gfCNCPoint4[26389] = {X -0.0949, Y 100.0187, Z -6.3333, A 0.000, B 0.000, C 0.000 }
gfCNCPoint4[26390] = {X -0.0672, Y 100.0699, Z -6.3333, A 0.000, B 0.000, C 0.000 }
gfCNCPoint4[26391] = {X -0.0148, Y 100.0951, Z -6.3333, A 0.000, B 0.000, C 0.000 }
gfCNCPoint4[26392] = {X 120.5926, Y 100.0951, Z -6.3333, A 0.000, B 0.000, C 0.000 }
gfCNCPoint4[26393] = {X 121.0614, Y 100.8813, Z -6.3333, A 0.000, B 0.000, C 0.000 }
gfCNCPoint4[26394] = {X 121.6687, Y 101.5661, Z -6.3333, A 0.000, B 0.000, C 0.000 }
gfCNCPoint4[26395] = {X 122.3932, Y 102.1254, Z -6.3333, A 0.000, B 0.000, C 0.000 }
gfCNCPoint4[26396] = {X 123.2095, Y 102.5397, Z -6.3333, A 0.000, B 0.000, C 0.000 }
gfCNCPoint4[26397] = {X 124.0887, Y 102.7942, Z -6.3333, A 0.000, B 0.000, C 0.000 }
gfCNCPoint4[26398] = {X 125.0000, Y 102.8800, Z -6.3333, A 0.000, B 0.000, C 0.000 }
gfCNCPoint4[26399] = {X 143.7791, Y 102.8800, Z -6.3333, A 0.000, B 0.000, C 0.000 }
gfCNCPoint4[26400] = {X 144.6904, Y 102.7942, Z -6.3333, A 0.000, B 0.000, C 0.000 }
gfCNCPoint4[26401] = {X 145.5696, Y 102.5397, Z -6.3333, A 0.000, B 0.000, C 0.000 }
gfCNCPoint4[26402] = {X 146.3859, Y 102.1254, Z -6.3333, A 0.000, B 0.000, C 0.000 }
gfCNCPoint4[26403] = {X 147.1104, Y 101.5661, Z -6.3333, A 0.000, B 0.000, C 0.000 }
gfCNCPoint4[26404] = {X 147.7177, Y 100.8813, Z -6.3333, A 0.000, B 0.000, C 0.000 }
gfCNCPoint4[26405] = {X 148.1865, Y 100.0951, Z -6.3333, A 0.000, B 0.000, C 0.000 }
gfCNCPoint4[26406] = {X 150.8385, Y 100.0951, Z -6.3333, A 0.000, B 0.000, C 0.000 }
gfCNCPoint4[26407] = {X 150.8385, Y 95.2951, Z -6.3333, A 0.000, B 0.000, C 0.000 }
gfCNCPoint4[26408] = {X 187.9256, Y 95.2951, Z -6.3333, A 0.000, B 0.000, C 0.000 }
gfCNCPoint4[26409] = {X 187.9777, Y 95.0990, Z -6.3333, A 0.000, B 0.000, C 0.000 }
gfCNCPoint4[26410] = {X 188.0352, Y 94.9045, Z -6.3333, A 0.000, B 0.000, C 0.000 }
gfCNCPoint4[26411] = {X 187.2619, Y 94.0602, Z -6.3333, A 0.000, B 0.000, C 0.000 }
gfCNCPoint4[26412] = {X 151.4055, Y 94.0602, Z -6.3333, A 0.000, B 0.000, C 0.000 }
gfCNCPoint4[26413] = {X 150.7064, Y 94.8347, Z -6.3333, A 0.000, B 0.000, C 0.000 }
gfCNCPoint4[26414] = {X 150.7762, Y 95.0638, Z -6.3333, A 0.000, B 0.000, C 0.000 }
gfCNCPoint4[26415] = {X 150.8385, Y 95.2951, Z -6.3333, A 0.000, B 0.000, C 0.000 }
gfCNCPoint4[26416] = {X 150.8385, Y 97.6951, Z -6.3333, A 0.000, B 0.000, C 0.000 }
gfCNCPoint4[26417] = {X 190.1070, Y 97.6951, Z -6.3333, A 0.000, B 0.000, C 0.000 }
gfCNCPoint4[26418] = {X 190.1070, Y 97.0659, Z -6.3333, A 0.000, B 0.000, C 0.000 }
gfCNCPoint4[26419] = {X 190.1938, Y 96.1495, Z -6.3333, A 0.000, B 0.000, C 0.000 }
gfCNCPoint4[26420] = {X 190.4511, Y 95.2657, Z -6.3333, A 0.000, B 0.000, C 0.000 }
gfCNCPoint4[26421] = {X 190.8699, Y 94.4460, Z -6.3333, A 0.000, B 0.000, C 0.000 }
gfCNCPoint4[26422] = {X 188.3182, Y 91.6602, Z -6.3333, A 0.000, B 0.000, C 0.000 }
gfCNCPoint4[26423] = {X 150.3387, Y 91.6602, Z -6.3333, A 0.000, B 0.000, C 0.000 }
gfCNCPoint4[26424] = {X 147.8644, Y 94.4015, Z -6.3333, A 0.000, B 0.000, C 0.000 }
gfCNCPoint4[26425] = {X 148.2989, Y 95.2324, Z -6.3333, A 0.000, B 0.000, C 0.000 }
gfCNCPoint4[26426] = {X 148.5670, Y 96.1308, Z -6.3333, A 0.000, B 0.000, C 0.000 }
gfCNCPoint4[26427] = {X 148.6591, Y 97.0639, Z -6.3333, A 0.000, B 0.000, C 0.000 }
gfCNCPoint4[26428] = {X 148.6591, Y 97.6951, Z -6.3333, A 0.000, B 0.000, C 0.000 }
gfCNCPoint4[26429] = {X 150.8385, Y 97.6951, Z -6.3333, A 0.000, B 0.000, C 0.000 }
gfCNCPoint4[26430] = {X 150.8385, Y 100.0951, Z -6.3333, A 0.000, B 0.000, C 0.000 }
gfCNCPoint4[26431] = {X 190.5796, Y 100.0951, Z -6.3333, A 0.000, B 0.000, C 0.000 }
gfCNCPoint4[26432] = {X 191.0483, Y 100.8813, Z -6.3333, A 0.000, B 0.000, C 0.000 }
gfCNCPoint4[26433] = {X 191.6557, Y 101.5661, Z -6.3333, A 0.000, B 0.000, C 0.000 }
gfCNCPoint4[26434] = {X 192.3802, Y 102.1254, Z -6.3333, A 0.000, B 0.000, C 0.000 }
gfCNCPoint4[26435] = {X 193.1964, Y 102.5397, Z -6.3333, A 0.000, B 0.000, C 0.000 }
gfCNCPoint4[26436] = {X 194.0757, Y 102.7942, Z -6.3333, A 0.000, B 0.000, C 0.000 }
gfCNCPoint4[26437] = {X 194.9870, Y 102.8800, Z -6.3333, A 0.000, B 0.000, C 0.000 }
gfCNCPoint4[26438] = {X 212.6141, Y 102.8800, Z -6.3333, A 0.000, B 0.000, C 0.000 }
gfCNCPoint4[26439] = {X 213.0066, Y 102.8642, Z -6.3333, A 0.000, B 0.000, C 0.000 }
gfCNCPoint4[26440] = {X 213.3966, Y 102.8169, Z -6.3333, A 0.000, B 0.000, C 0.000 }
gfCNCPoint4[26441] = {X 213.7865, Y 102.8642, Z -6.3333, A 0.000, B 0.000, C 0.000 }
gfCNCPoint4[26442] = {X 214.1790, Y 102.8800, Z -6.3333, A 0.000, B 0.000, C 0.000 }
gfCNCPoint4[26443] = {X 233.4798, Y 102.8800, Z -6.3333, A 0.000, B 0.000, C 0.000 }
gfCNCPoint4[26444] = {X 234.3911, Y 102.7942, Z -6.3333, A 0.000, B 0.000, C 0.000 }
gfCNCPoint4[26445] = {X 235.2703, Y 102.5397, Z -6.3333, A 0.000, B 0.000, C 0.000 }
gfCNCPoint4[26446] = {X 236.0865, Y 102.1254, Z -6.3333, A 0.000, B 0.000, C 0.000 }
gfCNCPoint4[26447] = {X 236.8111, Y 101.5661, Z -6.3333, A 0.000, B 0.000, C 0.000 }
gfCNCPoint4[26448] = {X 237.4184, Y 100.8813, Z -6.3333, A 0.000, B 0.000, C 0.000 }
gfCNCPoint4[26449] = {X 237.8872, Y 100.0951, Z -6.3333, A 0.000, B 0.000, C 0.000 }
gfCNCPoint4[26450] = {X 261.4782, Y 100.0951, Z -6.3333, A 0.000, B 0.000, C 0.000 }
gfCNCPoint4[26451] = {X 261.4782, Y 90.4951, Z -6.3333, A 0.000, B 0.000, C 0.000 }
gfCNCPoint4[26452] = {X 266.0961, Y 90.4951, Z -6.3333, A 0.000, B 0.000, C 0.000 }
gfCNCPoint4[26453] = {X 266.1751, Y 90.3748, Z -6.3333, A 0.000, B 0.000, C 0.000 }
gfCNCPoint4[26454] = {X 266.2556, Y 90.2554, Z -6.3333, A 0.000, B 0.000, C 0.000 }
gfCNCPoint4[26455] = {X 263.5100, Y 89.1791, Z -6.3333, A 0.000, B 0.000, C 0.000 }
gfCNCPoint4[26456] = {X 261.4782, Y 90.4951, Z -6.3333, A 0.000, B 0.000, C 0.000 }
gfCNCPoint4[26457] = {X 261.4782, Y 92.8951, Z -6.3333, A 0.000, B 0.000, C 0.000 }
gfCNCPoint4[26458] = {X 267.4973, Y 92.8951, Z -6.3333, A 0.000, B 0.000, C 0.000 }
gfCNCPoint4[26459] = {X 267.8429, Y 92.2376, Z -6.3333, A 0.000, B 0.000, C 0.000 }
gfCNCPoint4[26460] = {X 268.2378, Y 91.6085, Z -6.3333, A 0.000, B 0.000, C 0.000 }
gfCNCPoint4[26461] = {X 269.1700, Y 90.4463, Z -6.3333, A 0.000, B 0.000, C 0.000 }
gfCNCPoint4[26462] = {X 270.2694, Y 89.4409, Z -6.3333, A 0.000, B 0.000, C 0.000 }
gfCNCPoint4[26463] = {X 270.2694, Y 89.2510, Z -6.3333, A 0.000, B 0.000, C 0.000 }
gfCNCPoint4[26464] = {X 263.2391, Y 86.4951, Z -6.3333, A 0.000, B 0.000, C 0.000 }
gfCNCPoint4[26465] = {X 253.3583, Y 92.8951, Z -6.3333, A 0.000, B 0.000, C 0.000 }
gfCNCPoint4[26466] = {X 261.4782, Y 92.8951, Z -6.3333, A 0.000, B 0.000, C 0.000 }
gfCNCPoint4[26467] = {X 261.4782, Y 95.2951, Z -6.3333, A 0.000, B 0.000, C 0.000 }
gfCNCPoint4[26468] = {X 269.1714, Y 95.2951, Z -6.3333, A 0.000, B 0.000, C 0.000 }
gfCNCPoint4[26469] = {X 269.5515, Y 94.1745, Z -6.3333, A 0.000, B 0.000, C 0.000 }
gfCNCPoint4[26470] = {X 270.1082, Y 93.1303, Z -6.3333, A 0.000, B 0.000, C 0.000 }
gfCNCPoint4[26471] = {X 270.8267, Y 92.1901, Z -6.3333, A 0.000, B 0.000, C 0.000 }
gfCNCPoint4[26472] = {X 271.6880, Y 91.3787, Z -6.3333, A 0.000, B 0.000, C 0.000 }
gfCNCPoint4[26473] = {X 272.6694, Y 90.7176, Z -6.3333, A 0.000, B 0.000, C 0.000 }
gfCNCPoint4[26474] = {X 272.6694, Y 87.6139, Z -6.3333, A 0.000, B 0.000, C 0.000 }
gfCNCPoint4[26475] = {X 262.9682, Y 83.8111, Z -6.3333, A 0.000, B 0.000, C 0.000 }
gfCNCPoint4[26476] = {X 245.2384, Y 95.2951, Z -6.3333, A 0.000, B 0.000, C 0.000 }
gfCNCPoint4[26477] = {X 261.4782, Y 95.2951, Z -6.3333, A 0.000, B 0.000, C 0.000 }
gfCNCPoint4[26478] = {X 261.4782, Y 97.6951, Z -6.3333, A 0.000, B 0.000, C 0.000 }
gfCNCPoint4[26479] = {X 271.3527, Y 97.6951, Z -6.3333, A 0.000, B 0.000, C 0.000 }
gfCNCPoint4[26480] = {X 271.3529, Y 97.0186, Z -6.3333, A 0.000, B 0.000, C 0.000 }
gfCNCPoint4[26481] = {X 271.4810, Y 95.9545, Z -6.3333, A 0.000, B 0.000, C 0.000 }
gfCNCPoint4[26482] = {X 271.8382, Y 94.9440, Z -6.3333, A 0.000, B 0.000, C 0.000 }
gfCNCPoint4[26483] = {X 272.4073, Y 94.0359, Z -6.3333, A 0.000, B 0.000, C 0.000 }
gfCNCPoint4[26484] = {X 273.1610, Y 93.2739, Z -6.3333, A 0.000, B 0.000, C 0.000 }
gfCNCPoint4[26485] = {X 274.0629, Y 92.6949, Z -6.3333, A 0.000, B 0.000, C 0.000 }
gfCNCPoint4[26486] = {X 275.0694, Y 92.3266, Z -6.3333, A 0.000, B 0.000, C 0.000 }
gfCNCPoint4[26487] = {X 275.0694, Y 85.9769, Z -6.3333, A 0.000, B 0.000, C 0.000 }
gfCNCPoint4[26488] = {X 262.6992, Y 81.1278, Z -6.3333, A 0.000, B 0.000, C 0.000 }
gfCNCPoint4[26489] = {X 262.5795, Y 81.2034, Z -6.3333, A 0.000, B 0.000, C 0.000 }
gfCNCPoint4[26490] = {X 238.3588, Y 96.8917, Z -6.3333, A 0.000, B 0.000, C 0.000 }
gfCNCPoint4[26491] = {X 238.3598, Y 97.0659, Z -6.3333, A 0.000, B 0.000, C 0.000 }
gfCNCPoint4[26492] = {X 238.3598, Y 97.6951, Z -6.3333, A 0.000, B 0.000, C 0.000 }
gfCNCPoint4[26493] = {X 261.4782, Y 97.6951, Z -6.3333, A 0.000, B 0.000, C 0.000 }
gfCNCPoint4[26494] = {X 261.4782, Y 100.0951, Z -6.3333, A 0.000, B 0.000, C 0.000 }
gfCNCPoint4[26495] = {X 271.8253, Y 100.0951, Z -6.3333, A 0.000, B 0.000, C 0.000 }
gfCNCPoint4[26496] = {X 272.2941, Y 100.8813, Z -6.3333, A 0.000, B 0.000, C 0.000 }
gfCNCPoint4[26497] = {X 272.9014, Y 101.5661, Z -6.3333, A 0.000, B 0.000, C 0.000 }
gfCNCPoint4[26498] = {X 273.6259, Y 102.1254, Z -6.3333, A 0.000, B 0.000, C 0.000 }
gfCNCPoint4[26499] = {X 274.4422, Y 102.5397, Z -6.3333, A 0.000, B 0.000, C 0.000 }
gfCNCPoint4[26500] = {X 275.3214, Y 102.7942, Z -6.3333, A 0.000, B 0.000, C 0.000 }
gfCNCPoint4[26501] = {X 276.2327, Y 102.8800, Z -6.3333, A 0.000, B 0.000, C 0.000 }
gfCNCPoint4[26502] = {X 292.7731, Y 102.8800, Z -6.3333, A 0.000, B 0.000, C 0.000 }
gfCNCPoint4[26503] = {X 293.6844, Y 102.7942, Z -6.3333, A 0.000, B 0.000, C 0.000 }
gfCNCPoint4[26504] = {X 294.5636, Y 102.5397, Z -6.3333, A 0.000, B 0.000, C 0.000 }
gfCNCPoint4[26505] = {X 295.3798, Y 102.1254, Z -6.3333, A 0.000, B 0.000, C 0.000 }
gfCNCPoint4[26506] = {X 296.1044, Y 101.5661, Z -6.3333, A 0.000, B 0.000, C 0.000 }
gfCNCPoint4[26507] = {X 296.7117, Y 100.8813, Z -6.3333, A 0.000, B 0.000, C 0.000 }
gfCNCPoint4[26508] = {X 297.1805, Y 100.0951, Z -6.3333, A 0.000, B 0.000, C 0.000 }
gfCNCPoint4[26509] = {X 319.1325, Y 100.0951, Z -6.3333, A 0.000, B 0.000, C 0.000 }
gfCNCPoint4[26510] = {X 321.4361, Y 100.8683, Z -6.3333, A 0.000, B 0.000, C 0.000 }
gfCNCPoint4[26511] = {X 323.7823, Y 101.5005, Z -6.3333, A 0.000, B 0.000, C 0.000 }
gfCNCPoint4[26512] = {X 326.1626, Y 101.9893, Z -6.3333, A 0.000, B 0.000, C 0.000 }
gfCNCPoint4[26513] = {X 330.1025, Y 102.5988, Z -6.3333, A 0.000, B 0.000, C 0.000 }
gfCNCPoint4[26514] = {X 334.0644, Y 103.0432, Z -6.3333, A 0.000, B 0.000, C 0.000 }
gfCNCPoint4[26515] = {X 338.0414, Y 103.3217, Z -6.3333, A 0.000, B 0.000, C 0.000 }
gfCNCPoint4[26516] = {X 343.7798, Y 103.5423, Z -6.3333, A 0.000, B 0.000, C 0.000 }
gfCNCPoint4[26517] = {X 349.5223, Y 103.5874, Z -6.3333, A 0.000, B 0.000, C 0.000 }
gfCNCPoint4[26518] = {X 355.2635, Y 103.4570, Z -6.3333, A 0.000, B 0.000, C 0.000 }
gfCNCPoint4[26519] = {X 360.9980, Y 103.1512, Z -6.3333, A 0.000, B 0.000, C 0.000 }
gfCNCPoint4[26520] = {X 364.9923, Y 102.7834, Z -6.3333, A 0.000, B 0.000, C 0.000 }
gfCNCPoint4[26521] = {X 368.9636, Y 102.2191, Z -6.3333, A 0.000, B 0.000, C 0.000 }
gfCNCPoint4[26522] = {X 372.9022, Y 101.4595, Z -6.3333, A 0.000, B 0.000, C 0.000 }
gfCNCPoint4[26523] = {X 375.2297, Y 100.8564, Z -6.3333, A 0.000, B 0.000, C 0.000 }
gfCNCPoint4[26524] = {X 377.5103, Y 100.0951, Z -6.3333, A 0.000, B 0.000, C 0.000 }
gfCNCPoint4[26525] = {X 391.9986, Y 100.0951, Z -6.3333, A 0.000, B 0.000, C 0.000 }
gfCNCPoint4[26526] = {X 392.4673, Y 100.8813, Z -6.3333, A 0.000, B 0.000, C 0.000 }
gfCNCPoint4[26527] = {X 393.0747, Y 101.5661, Z -6.3333, A 0.000, B 0.000, C 0.000 }
gfCNCPoint4[26528] = {X 393.7992, Y 102.1254, Z -6.3333, A 0.000, B 0.000, C 0.000 }
gfCNCPoint4[26529] = {X 394.6154, Y 102.5397, Z -6.3333, A 0.000, B 0.000, C 0.000 }
gfCNCPoint4[26530] = {X 395.4947, Y 102.7942, Z -6.3333, A 0.000, B 0.000, C 0.000 }
gfCNCPoint4[26531] = {X 396.4059, Y 102.8800, Z -6.3333, A 0.000, B 0.000, C 0.000 }
gfCNCPoint4[26532] = {X 415.7067, Y 102.8800, Z -6.3333, A 0.000, B 0.000, C 0.000 }
gfCNCPoint4[26533] = {X 416.6180, Y 102.7942, Z -6.3333, A 0.000, B 0.000, C 0.000 }
gfCNCPoint4[26534] = {X 417.4972, Y 102.5397, Z -6.3333, A 0.000, B 0.000, C 0.000 }
gfCNCPoint4[26535] = {X 418.3135, Y 102.1254, Z -6.3333, A 0.000, B 0.000, C 0.000 }
gfCNCPoint4[26536] = {X 419.0380, Y 101.5661, Z -6.3333, A 0.000, B 0.000, C 0.000 }
gfCNCPoint4[26537] = {X 419.6453, Y 100.8813, Z -6.3333, A 0.000, B 0.000, C 0.000 }
gfCNCPoint4[26538] = {X 420.1141, Y 100.0951, Z -6.3333, A 0.000, B 0.000, C 0.000 }
gfCNCPoint4[26539] = {X 443.7037, Y 100.0951, Z -6.3333, A 0.000, B 0.000, C 0.000 }
gfCNCPoint4[26540] = {X 443.7037, Y 90.4951, Z -6.3333, A 0.000, B 0.000, C 0.000 }
gfCNCPoint4[26541] = {X 448.3230, Y 90.4951, Z -6.3333, A 0.000, B 0.000, C 0.000 }
gfCNCPoint4[26542] = {X 448.4020, Y 90.3748, Z -6.3333, A 0.000, B 0.000, C 0.000 }
gfCNCPoint4[26543] = {X 448.4825, Y 90.2554, Z -6.3333, A 0.000, B 0.000, C 0.000 }
gfCNCPoint4[26544] = {X 445.7359, Y 89.1787, Z -6.3333, A 0.000, B 0.000, C 0.000 }
gfCNCPoint4[26545] = {X 443.7037, Y 90.4951, Z -6.3333, A 0.000, B 0.000, C 0.000 }
gfCNCPoint4[26546] = {X 443.7037, Y 92.8951, Z -6.3333, A 0.000, B 0.000, C 0.000 }
gfCNCPoint4[26547] = {X 449.7242, Y 92.8951, Z -6.3333, A 0.000, B 0.000, C 0.000 }
gfCNCPoint4[26548] = {X 450.0698, Y 92.2376, Z -6.3333, A 0.000, B 0.000, C 0.000 }
gfCNCPoint4[26549] = {X 450.4647, Y 91.6084, Z -6.3333, A 0.000, B 0.000, C 0.000 }
gfCNCPoint4[26550] = {X 451.3969, Y 90.4463, Z -6.3333, A 0.000, B 0.000, C 0.000 }
gfCNCPoint4[26551] = {X 452.4963, Y 89.4409, Z -6.3333, A 0.000, B 0.000, C 0.000 }
gfCNCPoint4[26552] = {X 452.4963, Y 89.2510, Z -6.3333, A 0.000, B 0.000, C 0.000 }
gfCNCPoint4[26553] = {X 445.4649, Y 86.4947, Z -6.3333, A 0.000, B 0.000, C 0.000 }
gfCNCPoint4[26554] = {X 435.5843, Y 92.8951, Z -6.3333, A 0.000, B 0.000, C 0.000 }
gfCNCPoint4[26555] = {X 443.7037, Y 92.8951, Z -6.3333, A 0.000, B 0.000, C 0.000 }
gfCNCPoint4[26556] = {X 443.7037, Y 95.2951, Z -6.3333, A 0.000, B 0.000, C 0.000 }
gfCNCPoint4[26557] = {X 451.3983, Y 95.2951, Z -6.3333, A 0.000, B 0.000, C 0.000 }
gfCNCPoint4[26558] = {X 451.7784, Y 94.1745, Z -6.3333, A 0.000, B 0.000, C 0.000 }
gfCNCPoint4[26559] = {X 452.3351, Y 93.1303, Z -6.3333, A 0.000, B 0.000, C 0.000 }
gfCNCPoint4[26560] = {X 453.0536, Y 92.1901, Z -6.3333, A 0.000, B 0.000, C 0.000 }
gfCNCPoint4[26561] = {X 453.9149, Y 91.3787, Z -6.3333, A 0.000, B 0.000, C 0.000 }
gfCNCPoint4[26562] = {X 454.8963, Y 90.7176, Z -6.3333, A 0.000, B 0.000, C 0.000 }
gfCNCPoint4[26563] = {X 454.8963, Y 87.6139, Z -6.3333, A 0.000, B 0.000, C 0.000 }
gfCNCPoint4[26564] = {X 445.1940, Y 83.8106, Z -6.3333, A 0.000, B 0.000, C 0.000 }
gfCNCPoint4[26565] = {X 427.4649, Y 95.2951, Z -6.3333, A 0.000, B 0.000, C 0.000 }
gfCNCPoint4[26566] = {X 443.7037, Y 95.2951, Z -6.3333, A 0.000, B 0.000, C 0.000 }
gfCNCPoint4[26567] = {X 443.7037, Y 97.6951, Z -6.3333, A 0.000, B 0.000, C 0.000 }
gfCNCPoint4[26568] = {X 453.5796, Y 97.6951, Z -6.3333, A 0.000, B 0.000, C 0.000 }
gfCNCPoint4[26569] = {X 453.5796, Y 97.0659, Z -6.3333, A 0.000, B 0.000, C 0.000 }
gfCNCPoint4[26570] = {X 453.6990, Y 95.9930, Z -6.3333, A 0.000, B 0.000, C 0.000 }
gfCNCPoint4[26571] = {X 454.0514, Y 94.9725, Z -6.3333, A 0.000, B 0.000, C 0.000 }
gfCNCPoint4[26572] = {X 454.6196, Y 94.0545, Z -6.3333, A 0.000, B 0.000, C 0.000 }
gfCNCPoint4[26573] = {X 455.3757, Y 93.2839, Z -6.3333, A 0.000, B 0.000, C 0.000 }
gfCNCPoint4[26574] = {X 456.2827, Y 92.6984, Z -6.3333, A 0.000, B 0.000, C 0.000 }
gfCNCPoint4[26575] = {X 457.2963, Y 92.3266, Z -6.3333, A 0.000, B 0.000, C 0.000 }
gfCNCPoint4[26576] = {X 457.2963, Y 85.9769, Z -6.3333, A 0.000, B 0.000, C 0.000 }
gfCNCPoint4[26577] = {X 444.9230, Y 81.1266, Z -6.3333, A 0.000, B 0.000, C 0.000 }
gfCNCPoint4[26578] = {X 420.5857, Y 96.8917, Z -6.3333, A 0.000, B 0.000, C 0.000 }
gfCNCPoint4[26579] = {X 420.5867, Y 97.0659, Z -6.3333, A 0.000, B 0.000, C 0.000 }
gfCNCPoint4[26580] = {X 420.5867, Y 97.6951, Z -6.3333, A 0.000, B 0.000, C 0.000 }
gfCNCPoint4[26581] = {X 443.7037, Y 97.6951, Z -6.3333, A 0.000, B 0.000, C 0.000 }
gfCNCPoint4[26582] = {X 443.7037, Y 100.0951, Z -6.3333, A 0.000, B 0.000, C 0.000 }
gfCNCPoint4[26583] = {X 454.0522, Y 100.0951, Z -6.3333, A 0.000, B 0.000, C 0.000 }
gfCNCPoint4[26584] = {X 454.5210, Y 100.8813, Z -6.3333, A 0.000, B 0.000, C 0.000 }
gfCNCPoint4[26585] = {X 455.1283, Y 101.5661, Z -6.3333, A 0.000, B 0.000, C 0.000 }
gfCNCPoint4[26586] = {X 455.8529, Y 102.1254, Z -6.3333, A 0.000, B 0.000, C 0.000 }
gfCNCPoint4[26587] = {X 456.6691, Y 102.5397, Z -6.3333, A 0.000, B 0.000, C 0.000 }
gfCNCPoint4[26588] = {X 457.5483, Y 102.7942, Z -6.3333, A 0.000, B 0.000, C 0.000 }
gfCNCPoint4[26589] = {X 458.4596, Y 102.8800, Z -6.3333, A 0.000, B 0.000, C 0.000 }
gfCNCPoint4[26590] = {X 475.0000, Y 102.8800, Z -6.3333, A 0.000, B 0.000, C 0.000 }
gfCNCPoint4[26591] = {X 475.9113, Y 102.7942, Z -6.3333, A 0.000, B 0.000, C 0.000 }
gfCNCPoint4[26592] = {X 476.7905, Y 102.5397, Z -6.3333, A 0.000, B 0.000, C 0.000 }
gfCNCPoint4[26593] = {X 477.6068, Y 102.1254, Z -6.3333, A 0.000, B 0.000, C 0.000 }
gfCNCPoint4[26594] = {X 478.3313, Y 101.5661, Z -6.3333, A 0.000, B 0.000, C 0.000 }
gfCNCPoint4[26595] = {X 478.9386, Y 100.8813, Z -6.3333, A 0.000, B 0.000, C 0.000 }
gfCNCPoint4[26596] = {X 479.4074, Y 100.0951, Z -6.3333, A 0.000, B 0.000, C 0.000 }
gfCNCPoint4[26597] = {X 507.6813, Y 100.0951, Z -6.3333, A 0.000, B 0.000, C 0.000 }
gfCNCPoint4[26598] = {X 507.6813, Y 107.6951, Z -6.3333, A 0.000, B 0.000, C 0.000 }
gfCNCPoint4[26599] = {X 507.6813, Y 107.6951, Z -3.3333, A 0.000, B 0.000, C 0.000 }
gfCNCPoint4[26600] = {X 507.6813, Y 107.6951, Z 11.0000, A 0.000, B 0.000, C 0.000 }
gfCNCPoint4[26601] = {X 108.5567, Y 40.8981, Z 11.0000, A 0.000, B 0.000, C 0.000 }
gfCNCPoint4[26602] = {X 108.5567, Y 40.8981, Z -2.5000, A 0.000, B 0.000, C 0.000 }
gfCNCPoint4[26603] = {X 108.5567, Y 40.8981, Z -6.3333, A 0.000, B 0.000, C 0.000 }
gfCNCPoint4[26604] = {X 108.0683, Y 42.0917, Z -6.3333, A 0.000, B 0.000, C 0.000 }
gfCNCPoint4[26605] = {X 108.0971, Y 42.0416, Z -6.3333, A 0.000, B 0.000, C 0.000 }
gfCNCPoint4[26606] = {X 108.1266, Y 41.9919, Z -6.3333, A 0.000, B 0.000, C 0.000 }
gfCNCPoint4[26607] = {X 108.5492, Y 41.3813, Z -6.3333, A 0.000, B 0.000, C 0.000 }
gfCNCPoint4[26608] = {X 109.0453, Y 40.8286, Z -6.3333, A 0.000, B 0.000, C 0.000 }
gfCNCPoint4[26609] = {X 109.0452, Y 39.7044, Z -6.3333, A 0.000, B 0.000, C 0.000 }
gfCNCPoint4[26610] = {X 108.5567, Y 40.8981, Z -6.3333, A 0.000, B 0.000, C 0.000 }
gfCNCPoint4[26611] = {X 108.5567, Y 40.8981, Z -3.3333, A 0.000, B 0.000, C 0.000 }
gfCNCPoint4[26612] = {X 108.5567, Y 40.8981, Z 11.0000, A 0.000, B 0.000, C 0.000 }
gfCNCPoint4[26613] = {X 95.6826, Y 40.8720, Z 11.0000, A 0.000, B 0.000, C 0.000 }
gfCNCPoint4[26614] = {X 95.6826, Y 40.8720, Z -2.5000, A 0.000, B 0.000, C 0.000 }
gfCNCPoint4[26615] = {X 95.6826, Y 40.8720, Z -6.3333, A 0.000, B 0.000, C 0.000 }
gfCNCPoint4[26616] = {X 95.2117, Y 39.7204, Z -6.3333, A 0.000, B 0.000, C 0.000 }
gfCNCPoint4[26617] = {X 95.2117, Y 40.8683, Z -6.3333, A 0.000, B 0.000, C 0.000 }
gfCNCPoint4[26618] = {X 95.7310, Y 41.4066, Z -6.3333, A 0.000, B 0.000, C 0.000 }
gfCNCPoint4[26619] = {X 96.1535, Y 42.0237, Z -6.3333, A 0.000, B 0.000, C 0.000 }
gfCNCPoint4[26620] = {X 95.6826, Y 40.8720, Z -6.3333, A 0.000, B 0.000, C 0.000 }
gfCNCPoint4[26621] = {X 95.6826, Y 40.8720, Z -3.3333, A 0.000, B 0.000, C 0.000 }
gfCNCPoint4[26622] = {X 95.6826, Y 40.8720, Z 11.0000, A 0.000, B 0.000, C 0.000 }
gfCNCPoint4[26623] = {X -7.6966, Y 43.2876, Z 11.0000, A 0.000, B 0.000, C 0.000 }
gfCNCPoint4[26624] = {X -7.6966, Y 43.2876, Z -3.3333, A 0.000, B 0.000, C 0.000 }
gfCNCPoint4[26625] = {X -7.6966, Y 43.2876, Z -6.3333, A 0.000, B 0.000, C 0.000 }
gfCNCPoint4[26626] = {X -3.6966, Y 30.7997, Z -6.3333, A 0.000, B 0.000, C 0.000 }
gfCNCPoint4[26627] = {X -3.5210, Y 30.2839, Z -6.3333, A 0.000, B 0.000, C 0.000 }
gfCNCPoint4[26628] = {X -3.3266, Y 29.7750, Z -6.3333, A 0.000, B 0.000, C 0.000 }
gfCNCPoint4[26629] = {X -2.7036, Y 28.4548, Z -6.3333, A 0.000, B 0.000, C 0.000 }
gfCNCPoint4[26630] = {X -1.9098, Y 27.2297, Z -6.3333, A 0.000, B 0.000, C 0.000 }
gfCNCPoint4[26631] = {X -0.9594, Y 26.1216, Z -6.3333, A 0.000, B 0.000, C 0.000 }
gfCNCPoint4[26632] = {X 0.1304, Y 25.1504, Z -6.3333, A 0.000, B 0.000, C 0.000 }
gfCNCPoint4[26633] = {X 1.3402, Y 24.3335, Z -6.3333, A 0.000, B 0.000, C 0.000 }
gfCNCPoint4[26634] = {X 0.5798, Y 23.9233, Z -6.3333, A 0.000, B 0.000, C 0.000 }
gfCNCPoint4[26635] = {X -0.0859, Y 23.3723, Z -6.3333, A 0.000, B 0.000, C 0.000 }
gfCNCPoint4[26636] = {X -0.6310, Y 22.7019, Z -6.3333, A 0.000, B 0.000, C 0.000 }
gfCNCPoint4[26637] = {X -1.0345, Y 21.9379, Z -6.3333, A 0.000, B 0.000, C 0.000 }
gfCNCPoint4[26638] = {X -3.6458, Y 15.5423, Z -6.3333, A 0.000, B 0.000, C 0.000 }
gfCNCPoint4[26639] = {X -3.6717, Y 15.4773, Z -6.3333, A 0.000, B 0.000, C 0.000 }
gfCNCPoint4[26640] = {X -3.6966, Y 15.4118, Z -6.3333, A 0.000, B 0.000, C 0.000 }
gfCNCPoint4[26641] = {X -7.6966, Y 4.6481, Z -6.3333, A 0.000, B 0.000, C 0.000 }
gfCNCPoint4[26642] = {X -7.6966, Y 4.6481, Z -3.3333, A 0.000, B 0.000, C 0.000 }
gfCNCPoint4[26643] = {X -7.6966, Y 4.6481, Z 11.0000, A 0.000, B 0.000, C 0.000 }
gfCNCPoint4[26644] = {X -7.6966, Y 16.4129, Z 11.0000, A 0.000, B 0.000, C 0.000 }
gfCNCPoint4[26645] = {X -7.6966, Y 16.4129, Z -3.3333, A 0.000, B 0.000, C 0.000 }
gfCNCPoint4[26646] = {X -7.6966, Y 16.4129, Z -6.3333, A 0.000, B 0.000, C 0.000 }
gfCNCPoint4[26647] = {X -4.8866, Y 16.4129, Z -6.3333, A 0.000, B 0.000, C 0.000 }
gfCNCPoint4[26648] = {X -3.6966, Y 12.5940, Z -6.3333, A 0.000, B 0.000, C 0.000 }
gfCNCPoint4[26649] = {X -3.6606, Y 12.4836, Z -6.3333, A 0.000, B 0.000, C 0.000 }
gfCNCPoint4[26650] = {X -3.6216, Y 12.3743, Z -6.3333, A 0.000, B 0.000, C 0.000 }
gfCNCPoint4[26651] = {X -3.1667, Y 11.4829, Z -6.3333, A 0.000, B 0.000, C 0.000 }
gfCNCPoint4[26652] = {X -2.5189, Y 10.7201, Z -6.3333, A 0.000, B 0.000, C 0.000 }
gfCNCPoint4[26653] = {X -1.7129, Y 10.1268, Z -6.3333, A 0.000, B 0.000, C 0.000 }
gfCNCPoint4[26654] = {X -1.1156, Y 9.7861, Z -6.3333, A 0.000, B 0.000, C 0.000 }
gfCNCPoint4[26655] = {X -0.2327, Y 9.4056, Z -6.3333, A 0.000, B 0.000, C 0.000 }
gfCNCPoint4[26656] = {X 0.7125, Y 9.2298, Z -6.3333, A 0.000, B 0.000, C 0.000 }
gfCNCPoint4[26657] = {X 1.6731, Y 9.2674, Z -6.3333, A 0.000, B 0.000, C 0.000 }
gfCNCPoint4[26658] = {X 2.6017, Y 9.5165, Z -6.3333, A 0.000, B 0.000, C 0.000 }
gfCNCPoint4[26659] = {X 3.4887, Y 9.1197, Z -6.3333, A 0.000, B 0.000, C 0.000 }
gfCNCPoint4[26660] = {X 5.5656, Y 8.3372, Z -6.3333, A 0.000, B 0.000, C 0.000 }
gfCNCPoint4[26661] = {X 7.7065, Y 7.7514, Z -6.3333, A 0.000, B 0.000, C 0.000 }
gfCNCPoint4[26662] = {X 9.8925, Y 7.3676, Z -6.3333, A 0.000, B 0.000, C 0.000 }
gfCNCPoint4[26663] = {X 12.1048, Y 7.1891, Z -6.3333, A 0.000, B 0.000, C 0.000 }
gfCNCPoint4[26664] = {X 14.3241, Y 7.2174, Z -6.3333, A 0.000, B 0.000, C 0.000 }
gfCNCPoint4[26665] = {X 16.5311, Y 7.4523, Z -6.3333, A 0.000, B 0.000, C 0.000 }
gfCNCPoint4[26666] = {X 18.2665, Y 7.8078, Z -6.3333, A 0.000, B 0.000, C 0.000 }
gfCNCPoint4[26667] = {X 19.9569, Y 8.3374, Z -6.3333, A 0.000, B 0.000, C 0.000 }
gfCNCPoint4[26668] = {X 21.5849, Y 9.0356, Z -6.3333, A 0.000, B 0.000, C 0.000 }
gfCNCPoint4[26669] = {X 23.1337, Y 9.8953, Z -6.3333, A 0.000, B 0.000, C 0.000 }
gfCNCPoint4[26670] = {X 24.5873, Y 10.9077, Z -6.3333, A 0.000, B 0.000, C 0.000 }
gfCNCPoint4[26671] = {X 25.6728, Y 11.8567, Z -6.3333, A 0.000, B 0.000, C 0.000 }
gfCNCPoint4[26672] = {X 26.6464, Y 12.9200, Z -6.3333, A 0.000, B 0.000, C 0.000 }
gfCNCPoint4[26673] = {X 27.4963, Y 14.0846, Z -6.3333, A 0.000, B 0.000, C 0.000 }
gfCNCPoint4[26674] = {X 28.2121, Y 15.3362, Z -6.3333, A 0.000, B 0.000, C 0.000 }
gfCNCPoint4[26675] = {X 28.7849, Y 16.6593, Z -6.3333, A 0.000, B 0.000, C 0.000 }
gfCNCPoint4[26676] = {X 29.2597, Y 18.3155, Z -6.3333, A 0.000, B 0.000, C 0.000 }
gfCNCPoint4[26677] = {X 29.5416, Y 20.0152, Z -6.3333, A 0.000, B 0.000, C 0.000 }
gfCNCPoint4[26678] = {X 29.6266, Y 21.7360, Z -6.3333, A 0.000, B 0.000, C 0.000 }
gfCNCPoint4[26679] = {X 29.5138, Y 23.4552, Z -6.3333, A 0.000, B 0.000, C 0.000 }
gfCNCPoint4[26680] = {X 29.2045, Y 25.1502, Z -6.3333, A 0.000, B 0.000, C 0.000 }
gfCNCPoint4[26681] = {X 28.7622, Y 26.5966, Z -6.3333, A 0.000, B 0.000, C 0.000 }
gfCNCPoint4[26682] = {X 28.1369, Y 27.9738, Z -6.3333, A 0.000, B 0.000, C 0.000 }
gfCNCPoint4[26683] = {X 27.3390, Y 29.2587, Z -6.3333, A 0.000, B 0.000, C 0.000 }
gfCNCPoint4[26684] = {X 26.3819, Y 30.4299, Z -6.3333, A 0.000, B 0.000, C 0.000 }
gfCNCPoint4[26685] = {X 25.2817, Y 31.4678, Z -6.3333, A 0.000, B 0.000, C 0.000 }
gfCNCPoint4[26686] = {X 26.0855, Y 31.8100, Z -6.3333, A 0.000, B 0.000, C 0.000 }
gfCNCPoint4[26687] = {X 26.8041, Y 32.3069, Z -6.3333, A 0.000, B 0.000, C 0.000 }
gfCNCPoint4[26688] = {X 27.4080, Y 32.9382, Z -6.3333, A 0.000, B 0.000, C 0.000 }
gfCNCPoint4[26689] = {X 27.8726, Y 33.6781, Z -6.3333, A 0.000, B 0.000, C 0.000 }
gfCNCPoint4[26690] = {X 30.9100, Y 39.9530, Z -6.3333, A 0.000, B 0.000, C 0.000 }
gfCNCPoint4[26691] = {X 31.2306, Y 40.8622, Z -6.3333, A 0.000, B 0.000, C 0.000 }
gfCNCPoint4[26692] = {X 31.3415, Y 41.8197, Z -6.3333, A 0.000, B 0.000, C 0.000 }
gfCNCPoint4[26693] = {X 31.2374, Y 42.7781, Z -6.3333, A 0.000, B 0.000, C 0.000 }
gfCNCPoint4[26694] = {X 30.9234, Y 43.6895, Z -6.3333, A 0.000, B 0.000, C 0.000 }
gfCNCPoint4[26695] = {X 30.4150, Y 44.5085, Z -6.3333, A 0.000, B 0.000, C 0.000 }
gfCNCPoint4[26696] = {X 29.7377, Y 45.1945, Z -6.3333, A 0.000, B 0.000, C 0.000 }
gfCNCPoint4[26697] = {X 29.2017, Y 45.6279, Z -6.3333, A 0.000, B 0.000, C 0.000 }
gfCNCPoint4[26698] = {X 28.4977, Y 46.0916, Z -6.3333, A 0.000, B 0.000, C 0.000 }
gfCNCPoint4[26699] = {X 27.7173, Y 46.4101, Z -6.3333, A 0.000, B 0.000, C 0.000 }
gfCNCPoint4[26700] = {X 26.8900, Y 46.5715, Z -6.3333, A 0.000, B 0.000, C 0.000 }
gfCNCPoint4[26701] = {X 26.0470, Y 46.5696, Z -6.3333, A 0.000, B 0.000, C 0.000 }
gfCNCPoint4[26702] = {X 25.2204, Y 46.4044, Z -6.3333, A 0.000, B 0.000, C 0.000 }
gfCNCPoint4[26703] = {X 23.4202, Y 47.3538, Z -6.3333, A 0.000, B 0.000, C 0.000 }
gfCNCPoint4[26704] = {X 21.5586, Y 48.1762, Z -6.3333, A 0.000, B 0.000, C 0.000 }
gfCNCPoint4[26705] = {X 19.6445, Y 48.8676, Z -6.3333, A 0.000, B 0.000, C 0.000 }
gfCNCPoint4[26706] = {X 17.7045, Y 49.4154, Z -6.3333, A 0.000, B 0.000, C 0.000 }
gfCNCPoint4[26707] = {X 15.7237, Y 49.7892, Z -6.3333, A 0.000, B 0.000, C 0.000 }
gfCNCPoint4[26708] = {X 13.7175, Y 49.9863, Z -6.3333, A 0.000, B 0.000, C 0.000 }
gfCNCPoint4[26709] = {X 11.7018, Y 50.0050, Z -6.3333, A 0.000, B 0.000, C 0.000 }
gfCNCPoint4[26710] = {X 9.6923, Y 49.8453, Z -6.3333, A 0.000, B 0.000, C 0.000 }
gfCNCPoint4[26711] = {X 7.7049, Y 49.5083, Z -6.3333, A 0.000, B 0.000, C 0.000 }
gfCNCPoint4[26712] = {X 5.8036, Y 48.9872, Z -6.3333, A 0.000, B 0.000, C 0.000 }
gfCNCPoint4[26713] = {X 3.9769, Y 48.2460, Z -6.3333, A 0.000, B 0.000, C 0.000 }
gfCNCPoint4[26714] = {X 2.2501, Y 47.2949, Z -6.3333, A 0.000, B 0.000, C 0.000 }
gfCNCPoint4[26715] = {X 0.6472, Y 46.1472, Z -6.3333, A 0.000, B 0.000, C 0.000 }
gfCNCPoint4[26716] = {X -0.4851, Y 45.1293, Z -6.3333, A 0.000, B 0.000, C 0.000 }
gfCNCPoint4[26717] = {X -1.4909, Y 43.9861, Z -6.3333, A 0.000, B 0.000, C 0.000 }
gfCNCPoint4[26718] = {X -2.3562, Y 42.7332, Z -6.3333, A 0.000, B 0.000, C 0.000 }
gfCNCPoint4[26719] = {X -3.0694, Y 41.3879, Z -6.3333, A 0.000, B 0.000, C 0.000 }
gfCNCPoint4[26720] = {X -3.6205, Y 39.9685, Z -6.3333, A 0.000, B 0.000, C 0.000 }
gfCNCPoint4[26721] = {X -3.6592, Y 39.8465, Z -6.3333, A 0.000, B 0.000, C 0.000 }
gfCNCPoint4[26722] = {X -3.6966, Y 39.7241, Z -6.3333, A 0.000, B 0.000, C 0.000 }
gfCNCPoint4[26723] = {X -4.8487, Y 35.8936, Z -6.3333, A 0.000, B 0.000, C 0.000 }
gfCNCPoint4[26724] = {X -7.9947, Y 36.0064, Z -6.3333, A 0.000, B 0.000, C 0.000 }
gfCNCPoint4[26725] = {X -7.9947, Y 36.0064, Z -3.3333, A 0.000, B 0.000, C 0.000 }
gfCNCPoint4[26726] = {X -7.9947, Y 36.0064, Z 11.0000, A 0.000, B 0.000, C 0.000 }
gfCNCPoint4[26727] = {X 608.0000, Y 40.1192, Z 11.0000, A 0.000, B 0.000, C 0.000 }
gfCNCPoint4[26728] = {X 608.0000, Y 40.1192, Z -3.3333, A 0.000, B 0.000, C 0.000 }
gfCNCPoint4[26729] = {X 608.0000, Y 40.1192, Z -6.3333, A 0.000, B 0.000, C 0.000 }
gfCNCPoint4[26730] = {X 603.6966, Y 47.2355, Z -6.3333, A 0.000, B 0.000, C 0.000 }
gfCNCPoint4[26731] = {X 603.6634, Y 47.2895, Z -6.3333, A 0.000, B 0.000, C 0.000 }
gfCNCPoint4[26732] = {X 603.6294, Y 47.3430, Z -6.3333, A 0.000, B 0.000, C 0.000 }
gfCNCPoint4[26733] = {X 603.0931, Y 48.0158, Z -6.3333, A 0.000, B 0.000, C 0.000 }
gfCNCPoint4[26734] = {X 602.4340, Y 48.5690, Z -6.3333, A 0.000, B 0.000, C 0.000 }
gfCNCPoint4[26735] = {X 601.6784, Y 48.9806, Z -6.3333, A 0.000, B 0.000, C 0.000 }
gfCNCPoint4[26736] = {X 600.8562, Y 49.2343, Z -6.3333, A 0.000, B 0.000, C 0.000 }
gfCNCPoint4[26737] = {X 600.0000, Y 49.3200, Z -6.3333, A 0.000, B 0.000, C 0.000 }
gfCNCPoint4[26738] = {X 593.5565, Y 49.3200, Z -6.3333, A 0.000, B 0.000, C 0.000 }
gfCNCPoint4[26739] = {X 592.5952, Y 49.2117, Z -6.3333, A 0.000, B 0.000, C 0.000 }
gfCNCPoint4[26740] = {X 591.6822, Y 48.8922, Z -6.3333, A 0.000, B 0.000, C 0.000 }
gfCNCPoint4[26741] = {X 590.8631, Y 48.3775, Z -6.3333, A 0.000, B 0.000, C 0.000 }
gfCNCPoint4[26742] = {X 590.1790, Y 47.6935, Z -6.3333, A 0.000, B 0.000, C 0.000 }
gfCNCPoint4[26743] = {X 589.6643, Y 46.8744, Z -6.3333, A 0.000, B 0.000, C 0.000 }
gfCNCPoint4[26744] = {X 589.3448, Y 45.9613, Z -6.3333, A 0.000, B 0.000, C 0.000 }
gfCNCPoint4[26745] = {X 589.2365, Y 45.0000, Z -6.3333, A 0.000, B 0.000, C 0.000 }
gfCNCPoint4[26746] = {X 589.2365, Y 44.0647, Z -6.3333, A 0.000, B 0.000, C 0.000 }
gfCNCPoint4[26747] = {X 589.3405, Y 43.1363, Z -6.3333, A 0.000, B 0.000, C 0.000 }
gfCNCPoint4[26748] = {X 589.6399, Y 42.2515, Z -6.3333, A 0.000, B 0.000, C 0.000 }
gfCNCPoint4[26749] = {X 590.1209, Y 41.4507, Z -6.3333, A 0.000, B 0.000, C 0.000 }
gfCNCPoint4[26750] = {X 590.7616, Y 40.7709, Z -6.3333, A 0.000, B 0.000, C 0.000 }
gfCNCPoint4[26751] = {X 590.7623, Y 33.5322, Z -6.3333, A 0.000, B 0.000, C 0.000 }
gfCNCPoint4[26752] = {X 585.4453, Y 46.6524, Z -6.3333, A 0.000, B 0.000, C 0.000 }
gfCNCPoint4[26753] = {X 585.0755, Y 47.3550, Z -6.3333, A 0.000, B 0.000, C 0.000 }
gfCNCPoint4[26754] = {X 584.5834, Y 47.9780, Z -6.3333, A 0.000, B 0.000, C 0.000 }
gfCNCPoint4[26755] = {X 583.9856, Y 48.5004, Z -6.3333, A 0.000, B 0.000, C 0.000 }
gfCNCPoint4[26756] = {X 583.3023, Y 48.9046, Z -6.3333, A 0.000, B 0.000, C 0.000 }
gfCNCPoint4[26757] = {X 582.3585, Y 49.2242, Z -6.3333, A 0.000, B 0.000, C 0.000 }
gfCNCPoint4[26758] = {X 581.3666, Y 49.3191, Z -6.3333, A 0.000, B 0.000, C 0.000 }
gfCNCPoint4[26759] = {X 580.3794, Y 49.1842, Z -6.3333, A 0.000, B 0.000, C 0.000 }
gfCNCPoint4[26760] = {X 579.4493, Y 48.8268, Z -6.3333, A 0.000, B 0.000, C 0.000 }
gfCNCPoint4[26761] = {X 578.6259, Y 48.2657, Z -6.3333, A 0.000, B 0.000, C 0.000 }
gfCNCPoint4[26762] = {X 577.9529, Y 47.5309, Z -6.3333, A 0.000, B 0.000, C 0.000 }
gfCNCPoint4[26763] = {X 577.4662, Y 46.6615, Z -6.3333, A 0.000, B 0.000, C 0.000 }
gfCNCPoint4[26764] = {X 572.0196, Y 33.3431, Z -6.3333, A 0.000, B 0.000, C 0.000 }
gfCNCPoint4[26765] = {X 572.0225, Y 40.7728, Z -6.3333, A 0.000, B 0.000, C 0.000 }
gfCNCPoint4[26766] = {X 572.6595, Y 41.4437, Z -6.3333, A 0.000, B 0.000, C 0.000 }
gfCNCPoint4[26767] = {X 573.1391, Y 42.2348, Z -6.3333, A 0.000, B 0.000, C 0.000 }
gfCNCPoint4[26768] = {X 573.4393, Y 43.1098, Z -6.3333, A 0.000, B 0.000, C 0.000 }
gfCNCPoint4[26769] = {X 573.5463, Y 44.0287, Z -6.3333, A 0.000, B 0.000, C 0.000 }
gfCNCPoint4[26770] = {X 573.5464, Y 45.0000, Z -6.3333, A 0.000, B 0.000, C 0.000 }
gfCNCPoint4[26771] = {X 573.4381, Y 45.9613, Z -6.3333, A 0.000, B 0.000, C 0.000 }
gfCNCPoint4[26772] = {X 573.1186, Y 46.8744, Z -6.3333, A 0.000, B 0.000, C 0.000 }
gfCNCPoint4[26773] = {X 572.6039, Y 47.6935, Z -6.3333, A 0.000, B 0.000, C 0.000 }
gfCNCPoint4[26774] = {X 571.9199, Y 48.3775, Z -6.3333, A 0.000, B 0.000, C 0.000 }
gfCNCPoint4[26775] = {X 571.1008, Y 48.8922, Z -6.3333, A 0.000, B 0.000, C 0.000 }
gfCNCPoint4[26776] = {X 570.1877, Y 49.2117, Z -6.3333, A 0.000, B 0.000, C 0.000 }
gfCNCPoint4[26777] = {X 569.2264, Y 49.3200, Z -6.3333, A 0.000, B 0.000, C 0.000 }
gfCNCPoint4[26778] = {X 562.4443, Y 49.3200, Z -6.3333, A 0.000, B 0.000, C 0.000 }
gfCNCPoint4[26779] = {X 561.4830, Y 49.2117, Z -6.3333, A 0.000, B 0.000, C 0.000 }
gfCNCPoint4[26780] = {X 560.5699, Y 48.8922, Z -6.3333, A 0.000, B 0.000, C 0.000 }
gfCNCPoint4[26781] = {X 559.7508, Y 48.3775, Z -6.3333, A 0.000, B 0.000, C 0.000 }
gfCNCPoint4[26782] = {X 559.0668, Y 47.6935, Z -6.3333, A 0.000, B 0.000, C 0.000 }
gfCNCPoint4[26783] = {X 558.5521, Y 46.8744, Z -6.3333, A 0.000, B 0.000, C 0.000 }
gfCNCPoint4[26784] = {X 558.2326, Y 45.9613, Z -6.3333, A 0.000, B 0.000, C 0.000 }
gfCNCPoint4[26785] = {X 558.1243, Y 45.0000, Z -6.3333, A 0.000, B 0.000, C 0.000 }
gfCNCPoint4[26786] = {X 558.1243, Y 44.0648, Z -6.3333, A 0.000, B 0.000, C 0.000 }
gfCNCPoint4[26787] = {X 558.2280, Y 43.1360, Z -6.3333, A 0.000, B 0.000, C 0.000 }
gfCNCPoint4[26788] = {X 558.5277, Y 42.2508, Z -6.3333, A 0.000, B 0.000, C 0.000 }
gfCNCPoint4[26789] = {X 559.0095, Y 41.4500, Z -6.3333, A 0.000, B 0.000, C 0.000 }
gfCNCPoint4[26790] = {X 559.6512, Y 40.7706, Z -6.3333, A 0.000, B 0.000, C 0.000 }
gfCNCPoint4[26791] = {X 559.6512, Y 9.2296, Z -6.3333, A 0.000, B 0.000, C 0.000 }
gfCNCPoint4[26792] = {X 559.0130, Y 8.5587, Z -6.3333, A 0.000, B 0.000, C 0.000 }
gfCNCPoint4[26793] = {X 558.5325, Y 7.7672, Z -6.3333, A 0.000, B 0.000, C 0.000 }
gfCNCPoint4[26794] = {X 558.2317, Y 6.8915, Z -6.3333, A 0.000, B 0.000, C 0.000 }
gfCNCPoint4[26795] = {X 558.1245, Y 5.9718, Z -6.3333, A 0.000, B 0.000, C 0.000 }
gfCNCPoint4[26796] = {X 558.1243, Y 5.0000, Z -6.3333, A 0.000, B 0.000, C 0.000 }
gfCNCPoint4[26797] = {X 558.2326, Y 4.0387, Z -6.3333, A 0.000, B 0.000, C 0.000 }
gfCNCPoint4[26798] = {X 558.5521, Y 3.1256, Z -6.3333, A 0.000, B 0.000, C 0.000 }
gfCNCPoint4[26799] = {X 559.0668, Y 2.3065, Z -6.3333, A 0.000, B 0.000, C 0.000 }
gfCNCPoint4[26800] = {X 559.7508, Y 1.6225, Z -6.3333, A 0.000, B 0.000, C 0.000 }
gfCNCPoint4[26801] = {X 560.5699, Y 1.1078, Z -6.3333, A 0.000, B 0.000, C 0.000 }
gfCNCPoint4[26802] = {X 561.4830, Y 0.7883, Z -6.3333, A 0.000, B 0.000, C 0.000 }
gfCNCPoint4[26803] = {X 562.4443, Y 0.6800, Z -6.3333, A 0.000, B 0.000, C 0.000 }
gfCNCPoint4[26804] = {X 570.9376, Y 0.6800, Z -6.3333, A 0.000, B 0.000, C 0.000 }
gfCNCPoint4[26805] = {X 571.8988, Y 0.7883, Z -6.3333, A 0.000, B 0.000, C 0.000 }
gfCNCPoint4[26806] = {X 572.8119, Y 1.1078, Z -6.3333, A 0.000, B 0.000, C 0.000 }
gfCNCPoint4[26807] = {X 573.6310, Y 1.6225, Z -6.3333, A 0.000, B 0.000, C 0.000 }
gfCNCPoint4[26808] = {X 574.3151, Y 2.3065, Z -6.3333, A 0.000, B 0.000, C 0.000 }
gfCNCPoint4[26809] = {X 574.8297, Y 3.1256, Z -6.3333, A 0.000, B 0.000, C 0.000 }
gfCNCPoint4[26810] = {X 575.1492, Y 4.0387, Z -6.3333, A 0.000, B 0.000, C 0.000 }
gfCNCPoint4[26811] = {X 575.2576, Y 5.0000, Z -6.3333, A 0.000, B 0.000, C 0.000 }
gfCNCPoint4[26812] = {X 575.2576, Y 5.9342, Z -6.3333, A 0.000, B 0.000, C 0.000 }
gfCNCPoint4[26813] = {X 575.1835, Y 6.7303, Z -6.3333, A 0.000, B 0.000, C 0.000 }
gfCNCPoint4[26814] = {X 574.9641, Y 7.4991, Z -6.3333, A 0.000, B 0.000, C 0.000 }
gfCNCPoint4[26815] = {X 574.6068, Y 8.2142, Z -6.3333, A 0.000, B 0.000, C 0.000 }
gfCNCPoint4[26816] = {X 581.1910, Y 24.3691, Z -6.3333, A 0.000, B 0.000, C 0.000 }
gfCNCPoint4[26817] = {X 587.8456, Y 8.0939, Z -6.3333, A 0.000, B 0.000, C 0.000 }
gfCNCPoint4[26818] = {X 587.5316, Y 7.4228, Z -6.3333, A 0.000, B 0.000, C 0.000 }
gfCNCPoint4[26819] = {X 587.3369, Y 6.7081, Z -6.3333, A 0.000, B 0.000, C 0.000 }
gfCNCPoint4[26820] = {X 587.2671, Y 5.9705, Z -6.3333, A 0.000, B 0.000, C 0.000 }
gfCNCPoint4[26821] = {X 587.2670, Y 5.0000, Z -6.3333, A 0.000, B 0.000, C 0.000 }
gfCNCPoint4[26822] = {X 587.3753, Y 4.0387, Z -6.3333, A 0.000, B 0.000, C 0.000 }
gfCNCPoint4[26823] = {X 587.6948, Y 3.1256, Z -6.3333, A 0.000, B 0.000, C 0.000 }
gfCNCPoint4[26824] = {X 588.2094, Y 2.3065, Z -6.3333, A 0.000, B 0.000, C 0.000 }
gfCNCPoint4[26825] = {X 588.8935, Y 1.6225, Z -6.3333, A 0.000, B 0.000, C 0.000 }
gfCNCPoint4[26826] = {X 589.7126, Y 1.1078, Z -6.3333, A 0.000, B 0.000, C 0.000 }
gfCNCPoint4[26827] = {X 590.6257, Y 0.7883, Z -6.3333, A 0.000, B 0.000, C 0.000 }
gfCNCPoint4[26828] = {X 591.5870, Y 0.6800, Z -6.3333, A 0.000, B 0.000, C 0.000 }
gfCNCPoint4[26829] = {X 600.0000, Y 0.6800, Z -6.3333, A 0.000, B 0.000, C 0.000 }
gfCNCPoint4[26830] = {X 600.8562, Y 0.7657, Z -6.3333, A 0.000, B 0.000, C 0.000 }
gfCNCPoint4[26831] = {X 601.6784, Y 1.0194, Z -6.3333, A 0.000, B 0.000, C 0.000 }
gfCNCPoint4[26832] = {X 602.4340, Y 1.4310, Z -6.3333, A 0.000, B 0.000, C 0.000 }
gfCNCPoint4[26833] = {X 603.0931, Y 1.9842, Z -6.3333, A 0.000, B 0.000, C 0.000 }
gfCNCPoint4[26834] = {X 603.6294, Y 2.6570, Z -6.3333, A 0.000, B 0.000, C 0.000 }
gfCNCPoint4[26835] = {X 603.6634, Y 2.7105, Z -6.3333, A 0.000, B 0.000, C 0.000 }
gfCNCPoint4[26836] = {X 603.6966, Y 2.7645, Z -6.3333, A 0.000, B 0.000, C 0.000 }
gfCNCPoint4[26837] = {X 608.0000, Y 9.8807, Z -6.3333, A 0.000, B 0.000, C 0.000 }
gfCNCPoint4[26838] = {X 608.0000, Y 9.8807, Z -3.3333, A 0.000, B 0.000, C 0.000 }
gfCNCPoint4[26839] = {X 608.0000, Y 9.8807, Z 11.0000, A 0.000, B 0.000, C 0.000 }
gfCNCPoint4[26840] = {X -7.6966, Y 16.7868, Z 11.0000, A 0.000, B 0.000, C 0.000 }
gfCNCPoint4[26841] = {X -7.6966, Y 16.7868, Z -3.3333, A 0.000, B 0.000, C 0.000 }
gfCNCPoint4[26842] = {X -7.6966, Y 16.7868, Z -6.3333, A 0.000, B 0.000, C 0.000 }
gfCNCPoint4[26843] = {X -4.6242, Y 16.7868, Z -6.3333, A 0.000, B 0.000, C 0.000 }
gfCNCPoint4[26844] = {X -3.6966, Y 12.8959, Z -6.3333, A 0.000, B 0.000, C 0.000 }
gfCNCPoint4[26845] = {X -3.6292, Y 12.6467, Z -6.3333, A 0.000, B 0.000, C 0.000 }
gfCNCPoint4[26846] = {X -3.5467, Y 12.4022, Z -6.3333, A 0.000, B 0.000, C 0.000 }
gfCNCPoint4[26847] = {X -3.1002, Y 11.5273, Z -6.3333, A 0.000, B 0.000, C 0.000 }
gfCNCPoint4[26848] = {X -2.4643, Y 10.7786, Z -6.3333, A 0.000, B 0.000, C 0.000 }
gfCNCPoint4[26849] = {X -1.6733, Y 10.1963, Z -6.3333, A 0.000, B 0.000, C 0.000 }
gfCNCPoint4[26850] = {X -1.0760, Y 9.8556, Z -6.3333, A 0.000, B 0.000, C 0.000 }
gfCNCPoint4[26851] = {X -0.2015, Y 9.4797, Z -6.3333, A 0.000, B 0.000, C 0.000 }
gfCNCPoint4[26852] = {X 0.7349, Y 9.3084, Z -6.3333, A 0.000, B 0.000, C 0.000 }
gfCNCPoint4[26853] = {X 1.6859, Y 9.3503, Z -6.3333, A 0.000, B 0.000, C 0.000 }
gfCNCPoint4[26854] = {X 2.6036, Y 9.6033, Z -6.3333, A 0.000, B 0.000, C 0.000 }
gfCNCPoint4[26855] = {X 3.5209, Y 9.1930, Z -6.3333, A 0.000, B 0.000, C 0.000 }
gfCNCPoint4[26856] = {X 5.5908, Y 8.4131, Z -6.3333, A 0.000, B 0.000, C 0.000 }
gfCNCPoint4[26857] = {X 7.7243, Y 7.8294, Z -6.3333, A 0.000, B 0.000, C 0.000 }
gfCNCPoint4[26858] = {X 9.9029, Y 7.4469, Z -6.3333, A 0.000, B 0.000, C 0.000 }
gfCNCPoint4[26859] = {X 12.1077, Y 7.2691, Z -6.3333, A 0.000, B 0.000, C 0.000 }
gfCNCPoint4[26860] = {X 14.3195, Y 7.2973, Z -6.3333, A 0.000, B 0.000, C 0.000 }
gfCNCPoint4[26861] = {X 16.5190, Y 7.5314, Z -6.3333, A 0.000, B 0.000, C 0.000 }
gfCNCPoint4[26862] = {X 18.2464, Y 7.8852, Z -6.3333, A 0.000, B 0.000, C 0.000 }
gfCNCPoint4[26863] = {X 19.9291, Y 8.4124, Z -6.3333, A 0.000, B 0.000, C 0.000 }
gfCNCPoint4[26864] = {X 21.5496, Y 9.1074, Z -6.3333, A 0.000, B 0.000, C 0.000 }
gfCNCPoint4[26865] = {X 23.0914, Y 9.9632, Z -6.3333, A 0.000, B 0.000, C 0.000 }
gfCNCPoint4[26866] = {X 24.5384, Y 10.9709, Z -6.3333, A 0.000, B 0.000, C 0.000 }
gfCNCPoint4[26867] = {X 25.6170, Y 11.9141, Z -6.3333, A 0.000, B 0.000, C 0.000 }
gfCNCPoint4[26868] = {X 26.5846, Y 12.9708, Z -6.3333, A 0.000, B 0.000, C 0.000 }
gfCNCPoint4[26869] = {X 27.4293, Y 14.1283, Z -6.3333, A 0.000, B 0.000, C 0.000 }
gfCNCPoint4[26870] = {X 28.1406, Y 15.3721, Z -6.3333, A 0.000, B 0.000, C 0.000 }
gfCNCPoint4[26871] = {X 28.7098, Y 16.6870, Z -6.3333, A 0.000, B 0.000, C 0.000 }
gfCNCPoint4[26872] = {X 29.1820, Y 18.3342, Z -6.3333, A 0.000, B 0.000, C 0.000 }
gfCNCPoint4[26873] = {X 29.4621, Y 20.0246, Z -6.3333, A 0.000, B 0.000, C 0.000 }
gfCNCPoint4[26874] = {X 29.5466, Y 21.7360, Z -6.3333, A 0.000, B 0.000, C 0.000 }
gfCNCPoint4[26875] = {X 29.4343, Y 23.4459, Z -6.3333, A 0.000, B 0.000, C 0.000 }
gfCNCPoint4[26876] = {X 29.1267, Y 25.1315, Z -6.3333, A 0.000, B 0.000, C 0.000 }
gfCNCPoint4[26877] = {X 28.6767, Y 26.5964, Z -6.3333, A 0.000, B 0.000, C 0.000 }
gfCNCPoint4[26878] = {X 28.0377, Y 27.9893, Z -6.3333, A 0.000, B 0.000, C 0.000 }
gfCNCPoint4[26879] = {X 27.2208, Y 29.2859, Z -6.3333, A 0.000, B 0.000, C 0.000 }
gfCNCPoint4[26880] = {X 26.2403, Y 30.4637, Z -6.3333, A 0.000, B 0.000, C 0.000 }
gfCNCPoint4[26881] = {X 25.1133, Y 31.5021, Z -6.3333, A 0.000, B 0.000, C 0.000 }
gfCNCPoint4[26882] = {X 25.2528, Y 31.5426, Z -6.3333, A 0.000, B 0.000, C 0.000 }
gfCNCPoint4[26883] = {X 25.3908, Y 31.5879, Z -6.3333, A 0.000, B 0.000, C 0.000 }
gfCNCPoint4[26884] = {X 26.1382, Y 31.9318, Z -6.3333, A 0.000, B 0.000, C 0.000 }
gfCNCPoint4[26885] = {X 26.8050, Y 32.4136, Z -6.3333, A 0.000, B 0.000, C 0.000 }
gfCNCPoint4[26886] = {X 27.3663, Y 33.0150, Z -6.3333, A 0.000, B 0.000, C 0.000 }
gfCNCPoint4[26887] = {X 27.8009, Y 33.7136, Z -6.3333, A 0.000, B 0.000, C 0.000 }
gfCNCPoint4[26888] = {X 30.8380, Y 39.9879, Z -6.3333, A 0.000, B 0.000, C 0.000 }
gfCNCPoint4[26889] = {X 31.1526, Y 40.8802, Z -6.3333, A 0.000, B 0.000, C 0.000 }
gfCNCPoint4[26890] = {X 31.2615, Y 41.8200, Z -6.3333, A 0.000, B 0.000, C 0.000 }
gfCNCPoint4[26891] = {X 31.1593, Y 42.7606, Z -6.3333, A 0.000, B 0.000, C 0.000 }
gfCNCPoint4[26892] = {X 30.8511, Y 43.6551, Z -6.3333, A 0.000, B 0.000, C 0.000 }
gfCNCPoint4[26893] = {X 30.3522, Y 44.4590, Z -6.3333, A 0.000, B 0.000, C 0.000 }
gfCNCPoint4[26894] = {X 29.6874, Y 45.1323, Z -6.3333, A 0.000, B 0.000, C 0.000 }
gfCNCPoint4[26895] = {X 29.1514, Y 45.5657, Z -6.3333, A 0.000, B 0.000, C 0.000 }
gfCNCPoint4[26896] = {X 28.4543, Y 46.0240, Z -6.3333, A 0.000, B 0.000, C 0.000 }
gfCNCPoint4[26897] = {X 27.6812, Y 46.3374, Z -6.3333, A 0.000, B 0.000, C 0.000 }
gfCNCPoint4[26898] = {X 26.8618, Y 46.4938, Z -6.3333, A 0.000, B 0.000, C 0.000 }
gfCNCPoint4[26899] = {X 26.0276, Y 46.4871, Z -6.3333, A 0.000, B 0.000, C 0.000 }
gfCNCPoint4[26900] = {X 25.2108, Y 46.3178, Z -6.3333, A 0.000, B 0.000, C 0.000 }
gfCNCPoint4[26901] = {X 23.4061, Y 47.2717, Z -6.3333, A 0.000, B 0.000, C 0.000 }
gfCNCPoint4[26902] = {X 21.5394, Y 48.0977, Z -6.3333, A 0.000, B 0.000, C 0.000 }
gfCNCPoint4[26903] = {X 19.6197, Y 48.7916, Z -6.3333, A 0.000, B 0.000, C 0.000 }
gfCNCPoint4[26904] = {X 17.6865, Y 49.3374, Z -6.3333, A 0.000, B 0.000, C 0.000 }
gfCNCPoint4[26905] = {X 15.7125, Y 49.7100, Z -6.3333, A 0.000, B 0.000, C 0.000 }
gfCNCPoint4[26906] = {X 13.7134, Y 49.9064, Z -6.3333, A 0.000, B 0.000, C 0.000 }
gfCNCPoint4[26907] = {X 11.7047, Y 49.9251, Z -6.3333, A 0.000, B 0.000, C 0.000 }
gfCNCPoint4[26908] = {X 9.7022, Y 49.7659, Z -6.3333, A 0.000, B 0.000, C 0.000 }
gfCNCPoint4[26909] = {X 7.7217, Y 49.4301, Z -6.3333, A 0.000, B 0.000, C 0.000 }
gfCNCPoint4[26910] = {X 5.8294, Y 48.9115, Z -6.3333, A 0.000, B 0.000, C 0.000 }
gfCNCPoint4[26911] = {X 4.0113, Y 48.1738, Z -6.3333, A 0.000, B 0.000, C 0.000 }
gfCNCPoint4[26912] = {X 2.2926, Y 47.2272, Z -6.3333, A 0.000, B 0.000, C 0.000 }
gfCNCPoint4[26913] = {X 0.6974, Y 46.0849, Z -6.3333, A 0.000, B 0.000, C 0.000 }
gfCNCPoint4[26914] = {X -0.4281, Y 45.0732, Z -6.3333, A 0.000, B 0.000, C 0.000 }
gfCNCPoint4[26915] = {X -1.4277, Y 43.9370, Z -6.3333, A 0.000, B 0.000, C 0.000 }
gfCNCPoint4[26916] = {X -2.2878, Y 42.6918, Z -6.3333, A 0.000, B 0.000, C 0.000 }
gfCNCPoint4[26917] = {X -2.9966, Y 41.3547, Z -6.3333, A 0.000, B 0.000, C 0.000 }
gfCNCPoint4[26918] = {X -3.5444, Y 39.9440, Z -6.3333, A 0.000, B 0.000, C 0.000 }
gfCNCPoint4[26919] = {X -3.6231, Y 39.6908, Z -6.3333, A 0.000, B 0.000, C 0.000 }
gfCNCPoint4[26920] = {X -3.6966, Y 39.4361, Z -6.3333, A 0.000, B 0.000, C 0.000 }
gfCNCPoint4[26921] = {X -4.7668, Y 35.5820, Z -6.3333, A 0.000, B 0.000, C 0.000 }
gfCNCPoint4[26922] = {X -8.0043, Y 35.6326, Z -6.3333, A 0.000, B 0.000, C 0.000 }
gfCNCPoint4[26923] = {X -8.0043, Y 35.6326, Z -3.3333, A 0.000, B 0.000, C 0.000 }
gfCNCPoint4[26924] = {X -8.0043, Y 35.6326, Z 11.0000, A 0.000, B 0.000, C 0.000 }
gfCNCPoint4[26925] = {X -7.6966, Y 17.3020, Z 11.0000, A 0.000, B 0.000, C 0.000 }
gfCNCPoint4[26926] = {X -7.6966, Y 17.3020, Z -3.3333, A 0.000, B 0.000, C 0.000 }
gfCNCPoint4[26927] = {X -7.6966, Y 17.3020, Z -6.3333, A 0.000, B 0.000, C 0.000 }
gfCNCPoint4[26928] = {X -4.2187, Y 17.3020, Z -6.3333, A 0.000, B 0.000, C 0.000 }
gfCNCPoint4[26929] = {X -3.6966, Y 13.3362, Z -6.3333, A 0.000, B 0.000, C 0.000 }
gfCNCPoint4[26930] = {X -3.6097, Y 12.8768, Z -6.3333, A 0.000, B 0.000, C 0.000 }
gfCNCPoint4[26931] = {X -3.4717, Y 12.4300, Z -6.3333, A 0.000, B 0.000, C 0.000 }
gfCNCPoint4[26932] = {X -3.0336, Y 11.5716, Z -6.3333, A 0.000, B 0.000, C 0.000 }
gfCNCPoint4[26933] = {X -2.4098, Y 10.8371, Z -6.3333, A 0.000, B 0.000, C 0.000 }
gfCNCPoint4[26934] = {X -1.6337, Y 10.2658, Z -6.3333, A 0.000, B 0.000, C 0.000 }
gfCNCPoint4[26935] = {X -1.0364, Y 9.9250, Z -6.3333, A 0.000, B 0.000, C 0.000 }
gfCNCPoint4[26936] = {X -0.1702, Y 9.5538, Z -6.3333, A 0.000, B 0.000, C 0.000 }
gfCNCPoint4[26937] = {X 0.7573, Y 9.3871, Z -6.3333, A 0.000, B 0.000, C 0.000 }
gfCNCPoint4[26938] = {X 1.6985, Y 9.4334, Z -6.3333, A 0.000, B 0.000, C 0.000 }
gfCNCPoint4[26939] = {X 2.6051, Y 9.6903, Z -6.3333, A 0.000, B 0.000, C 0.000 }
gfCNCPoint4[26940] = {X 3.5530, Y 9.2662, Z -6.3333, A 0.000, B 0.000, C 0.000 }
gfCNCPoint4[26941] = {X 5.6159, Y 8.4891, Z -6.3333, A 0.000, B 0.000, C 0.000 }
gfCNCPoint4[26942] = {X 7.7422, Y 7.9074, Z -6.3333, A 0.000, B 0.000, C 0.000 }
gfCNCPoint4[26943] = {X 9.9134, Y 7.5263, Z -6.3333, A 0.000, B 0.000, C 0.000 }
gfCNCPoint4[26944] = {X 12.1106, Y 7.3490, Z -6.3333, A 0.000, B 0.000, C 0.000 }
gfCNCPoint4[26945] = {X 14.3148, Y 7.3772, Z -6.3333, A 0.000, B 0.000, C 0.000 }
gfCNCPoint4[26946] = {X 16.5068, Y 7.6105, Z -6.3333, A 0.000, B 0.000, C 0.000 }
gfCNCPoint4[26947] = {X 18.2263, Y 7.9627, Z -6.3333, A 0.000, B 0.000, C 0.000 }
gfCNCPoint4[26948] = {X 19.9013, Y 8.4874, Z -6.3333, A 0.000, B 0.000, C 0.000 }
gfCNCPoint4[26949] = {X 21.5144, Y 9.1792, Z -6.3333, A 0.000, B 0.000, C 0.000 }
gfCNCPoint4[26950] = {X 23.0490, Y 10.0311, Z -6.3333, A 0.000, B 0.000, C 0.000 }
gfCNCPoint4[26951] = {X 24.4894, Y 11.0342, Z -6.3333, A 0.000, B 0.000, C 0.000 }
gfCNCPoint4[26952] = {X 25.5613, Y 11.9715, Z -6.3333, A 0.000, B 0.000, C 0.000 }
gfCNCPoint4[26953] = {X 26.5228, Y 13.0217, Z -6.3333, A 0.000, B 0.000, C 0.000 }
gfCNCPoint4[26954] = {X 27.3622, Y 14.1719, Z -6.3333, A 0.000, B 0.000, C 0.000 }
gfCNCPoint4[26955] = {X 28.0691, Y 15.4079, Z -6.3333, A 0.000, B 0.000, C 0.000 }
gfCNCPoint4[26956] = {X 28.6347, Y 16.7147, Z -6.3333, A 0.000, B 0.000, C 0.000 }
gfCNCPoint4[26957] = {X 29.1042, Y 18.3528, Z -6.3333, A 0.000, B 0.000, C 0.000 }
gfCNCPoint4[26958] = {X 29.3827, Y 20.0340, Z -6.3333, A 0.000, B 0.000, C 0.000 }
gfCNCPoint4[26959] = {X 29.4666, Y 21.7361, Z -6.3333, A 0.000, B 0.000, C 0.000 }
gfCNCPoint4[26960] = {X 29.3549, Y 23.4365, Z -6.3333, A 0.000, B 0.000, C 0.000 }
gfCNCPoint4[26961] = {X 29.0489, Y 25.1129, Z -6.3333, A 0.000, B 0.000, C 0.000 }
gfCNCPoint4[26962] = {X 28.5905, Y 26.5979, Z -6.3333, A 0.000, B 0.000, C 0.000 }
gfCNCPoint4[26963] = {X 27.9365, Y 28.0078, Z -6.3333, A 0.000, B 0.000, C 0.000 }
gfCNCPoint4[26964] = {X 27.0989, Y 29.3169, Z -6.3333, A 0.000, B 0.000, C 0.000 }
gfCNCPoint4[26965] = {X 26.0929, Y 30.5015, Z -6.3333, A 0.000, B 0.000, C 0.000 }
gfCNCPoint4[26966] = {X 24.9367, Y 31.5402, Z -6.3333, A 0.000, B 0.000, C 0.000 }
gfCNCPoint4[26967] = {X 25.1523, Y 31.5961, Z -6.3333, A 0.000, B 0.000, C 0.000 }
gfCNCPoint4[26968] = {X 25.3646, Y 31.6635, Z -6.3333, A 0.000, B 0.000, C 0.000 }
gfCNCPoint4[26969] = {X 26.0978, Y 32.0009, Z -6.3333, A 0.000, B 0.000, C 0.000 }
gfCNCPoint4[26970] = {X 26.7521, Y 32.4736, Z -6.3333, A 0.000, B 0.000, C 0.000 }
gfCNCPoint4[26971] = {X 27.3028, Y 33.0637, Z -6.3333, A 0.000, B 0.000, C 0.000 }
gfCNCPoint4[26972] = {X 27.7292, Y 33.7491, Z -6.3333, A 0.000, B 0.000, C 0.000 }
gfCNCPoint4[26973] = {X 30.7660, Y 40.0227, Z -6.3333, A 0.000, B 0.000, C 0.000 }
gfCNCPoint4[26974] = {X 31.0747, Y 40.8982, Z -6.3333, A 0.000, B 0.000, C 0.000 }
gfCNCPoint4[26975] = {X 31.1815, Y 41.8203, Z -6.3333, A 0.000, B 0.000, C 0.000 }
gfCNCPoint4[26976] = {X 31.0813, Y 42.7431, Z -6.3333, A 0.000, B 0.000, C 0.000 }
gfCNCPoint4[26977] = {X 30.7789, Y 43.6208, Z -6.3333, A 0.000, B 0.000, C 0.000 }
gfCNCPoint4[26978] = {X 30.2893, Y 44.4095, Z -6.3333, A 0.000, B 0.000, C 0.000 }
gfCNCPoint4[26979] = {X 29.6371, Y 45.0700, Z -6.3333, A 0.000, B 0.000, C 0.000 }
gfCNCPoint4[26980] = {X 29.1011, Y 45.5035, Z -6.3333, A 0.000, B 0.000, C 0.000 }
gfCNCPoint4[26981] = {X 28.4110, Y 45.9564, Z -6.3333, A 0.000, B 0.000, C 0.000 }
gfCNCPoint4[26982] = {X 27.6452, Y 46.2646, Z -6.3333, A 0.000, B 0.000, C 0.000 }
gfCNCPoint4[26983] = {X 26.8338, Y 46.4159, Z -6.3333, A 0.000, B 0.000, C 0.000 }
gfCNCPoint4[26984] = {X 26.0084, Y 46.4046, Z -6.3333, A 0.000, B 0.000, C 0.000 }
gfCNCPoint4[26985] = {X 25.2014, Y 46.2309, Z -6.3333, A 0.000, B 0.000, C 0.000 }
gfCNCPoint4[26986] = {X 23.3922, Y 47.1896, Z -6.3333, A 0.000, B 0.000, C 0.000 }
gfCNCPoint4[26987] = {X 21.5203, Y 48.0191, Z -6.3333, A 0.000, B 0.000, C 0.000 }
gfCNCPoint4[26988] = {X 19.5948, Y 48.7155, Z -6.3333, A 0.000, B 0.000, C 0.000 }
gfCNCPoint4[26989] = {X 17.6684, Y 49.2595, Z -6.3333, A 0.000, B 0.000, C 0.000 }
gfCNCPoint4[26990] = {X 15.7013, Y 49.6308, Z -6.3333, A 0.000, B 0.000, C 0.000 }
gfCNCPoint4[26991] = {X 13.7092, Y 49.8265, Z -6.3333, A 0.000, B 0.000, C 0.000 }
gfCNCPoint4[26992] = {X 11.7075, Y 49.8451, Z -6.3333, A 0.000, B 0.000, C 0.000 }
gfCNCPoint4[26993] = {X 9.7120, Y 49.6865, Z -6.3333, A 0.000, B 0.000, C 0.000 }
gfCNCPoint4[26994] = {X 7.7384, Y 49.3518, Z -6.3333, A 0.000, B 0.000, C 0.000 }
gfCNCPoint4[26995] = {X 5.8551, Y 48.8357, Z -6.3333, A 0.000, B 0.000, C 0.000 }
gfCNCPoint4[26996] = {X 4.0456, Y 48.1015, Z -6.3333, A 0.000, B 0.000, C 0.000 }
gfCNCPoint4[26997] = {X 2.3352, Y 47.1594, Z -6.3333, A 0.000, B 0.000, C 0.000 }
gfCNCPoint4[26998] = {X 0.7475, Y 46.0225, Z -6.3333, A 0.000, B 0.000, C 0.000 }
gfCNCPoint4[26999] = {X -0.3711, Y 45.0171, Z -6.3333, A 0.000, B 0.000, C 0.000 }
gfCNCPoint4[27000] = {X -1.3646, Y 43.8879, Z -6.3333, A 0.000, B 0.000, C 0.000 }
gfCNCPoint4[27001] = {X -2.2194, Y 42.6504, Z -6.3333, A 0.000, B 0.000, C 0.000 }
gfCNCPoint4[27002] = {X -2.9238, Y 41.3215, Z -6.3333, A 0.000, B 0.000, C 0.000 }
gfCNCPoint4[27003] = {X -3.4682, Y 39.9194, Z -6.3333, A 0.000, B 0.000, C 0.000 }
gfCNCPoint4[27004] = {X -3.5888, Y 39.5235, Z -6.3333, A 0.000, B 0.000, C 0.000 }
gfCNCPoint4[27005] = {X -3.6966, Y 39.1240, Z -6.3333, A 0.000, B 0.000, C 0.000 }
gfCNCPoint4[27006] = {X -4.6764, Y 35.2458, Z -6.3333, A 0.000, B 0.000, C 0.000 }
gfCNCPoint4[27007] = {X -8.0062, Y 35.2244, Z -6.3333, A 0.000, B 0.000, C 0.000 }
gfCNCPoint4[27008] = {X -8.0062, Y 35.2244, Z -3.3333, A 0.000, B 0.000, C 0.000 }
gfCNCPoint4[27009] = {X -8.0062, Y 35.2244, Z 11.0000, A 0.000, B 0.000, C 0.000 }
gfCNCPoint4[27010] = {X -7.9988, Y 34.8079, Z 11.0000, A 0.000, B 0.000, C 0.000 }
gfCNCPoint4[27011] = {X -7.9988, Y 34.8079, Z -3.3333, A 0.000, B 0.000, C 0.000 }
gfCNCPoint4[27012] = {X -7.9988, Y 34.8079, Z -6.3333, A 0.000, B 0.000, C 0.000 }
gfCNCPoint4[27013] = {X -4.8506, Y 34.8991, Z -6.3333, A 0.000, B 0.000, C 0.000 }
gfCNCPoint4[27014] = {X -3.6966, Y 31.0692, Z -6.3333, A 0.000, B 0.000, C 0.000 }
gfCNCPoint4[27015] = {X -3.6591, Y 30.9465, Z -6.3333, A 0.000, B 0.000, C 0.000 }
gfCNCPoint4[27016] = {X -3.6204, Y 30.8241, Z -6.3333, A 0.000, B 0.000, C 0.000 }
gfCNCPoint4[27017] = {X -3.4459, Y 30.3116, Z -6.3333, A 0.000, B 0.000, C 0.000 }
gfCNCPoint4[27018] = {X -3.2528, Y 29.8059, Z -6.3333, A 0.000, B 0.000, C 0.000 }
gfCNCPoint4[27019] = {X -2.6182, Y 28.4661, Z -6.3333, A 0.000, B 0.000, C 0.000 }
gfCNCPoint4[27020] = {X -1.8065, Y 27.2255, Z -6.3333, A 0.000, B 0.000, C 0.000 }
gfCNCPoint4[27021] = {X -0.8329, Y 26.1075, Z -6.3333, A 0.000, B 0.000, C 0.000 }
gfCNCPoint4[27022] = {X 0.2844, Y 25.1331, Z -6.3333, A 0.000, B 0.000, C 0.000 }
gfCNCPoint4[27023] = {X 1.5243, Y 24.3205, Z -6.3333, A 0.000, B 0.000, C 0.000 }
gfCNCPoint4[27024] = {X 0.7360, Y 23.9296, Z -6.3333, A 0.000, B 0.000, C 0.000 }
gfCNCPoint4[27025] = {X 0.0432, Y 23.3871, Z -6.3333, A 0.000, B 0.000, C 0.000 }
gfCNCPoint4[27026] = {X -0.5253, Y 22.7155, Z -6.3333, A 0.000, B 0.000, C 0.000 }
gfCNCPoint4[27027] = {X -0.9460, Y 21.9427, Z -6.3333, A 0.000, B 0.000, C 0.000 }
gfCNCPoint4[27028] = {X -3.6216, Y 15.3840, Z -6.3333, A 0.000, B 0.000, C 0.000 }
gfCNCPoint4[27029] = {X -3.6606, Y 15.2746, Z -6.3333, A 0.000, B 0.000, C 0.000 }
gfCNCPoint4[27030] = {X -3.6966, Y 15.1643, Z -6.3333, A 0.000, B 0.000, C 0.000 }
gfCNCPoint4[27031] = {X -4.8866, Y 11.3454, Z -6.3333, A 0.000, B 0.000, C 0.000 }
gfCNCPoint4[27032] = {X -7.6966, Y 11.3454, Z -6.3333, A 0.000, B 0.000, C 0.000 }
gfCNCPoint4[27033] = {X -7.6966, Y 11.3454, Z -3.3333, A 0.000, B 0.000, C 0.000 }
gfCNCPoint4[27034] = {X -7.6966, Y 11.3454, Z 11.0000, A 0.000, B 0.000, C 0.000 }
gfCNCPoint4[27035] = {X -8.0058, Y 35.1770, Z 11.0000, A 0.000, B 0.000, C 0.000 }
gfCNCPoint4[27036] = {X -8.0058, Y 35.1770, Z -3.3333, A 0.000, B 0.000, C 0.000 }
gfCNCPoint4[27037] = {X -8.0058, Y 35.1770, Z -6.3333, A 0.000, B 0.000, C 0.000 }
gfCNCPoint4[27038] = {X -4.7792, Y 35.2061, Z -6.3333, A 0.000, B 0.000, C 0.000 }
gfCNCPoint4[27039] = {X -3.6966, Y 31.3553, Z -6.3333, A 0.000, B 0.000, C 0.000 }
gfCNCPoint4[27040] = {X -3.6227, Y 31.1012, Z -6.3333, A 0.000, B 0.000, C 0.000 }
gfCNCPoint4[27041] = {X -3.5443, Y 30.8485, Z -6.3333, A 0.000, B 0.000, C 0.000 }
gfCNCPoint4[27042] = {X -3.3706, Y 30.3386, Z -6.3333, A 0.000, B 0.000, C 0.000 }
gfCNCPoint4[27043] = {X -3.1785, Y 29.8355, Z -6.3333, A 0.000, B 0.000, C 0.000 }
gfCNCPoint4[27044] = {X -2.5646, Y 28.5342, Z -6.3333, A 0.000, B 0.000, C 0.000 }
gfCNCPoint4[27045] = {X -1.7824, Y 27.3266, Z -6.3333, A 0.000, B 0.000, C 0.000 }
gfCNCPoint4[27046] = {X -0.8459, Y 26.2343, Z -6.3333, A 0.000, B 0.000, C 0.000 }
gfCNCPoint4[27047] = {X 0.2283, Y 25.2770, Z -6.3333, A 0.000, B 0.000, C 0.000 }
gfCNCPoint4[27048] = {X 1.4207, Y 24.4718, Z -6.3333, A 0.000, B 0.000, C 0.000 }
gfCNCPoint4[27049] = {X 1.5695, Y 24.3868, Z -6.3333, A 0.000, B 0.000, C 0.000 }
gfCNCPoint4[27050] = {X 1.7197, Y 24.3042, Z -6.3333, A 0.000, B 0.000, C 0.000 }
gfCNCPoint4[27051] = {X 0.8922, Y 23.9311, Z -6.3333, A 0.000, B 0.000, C 0.000 }
gfCNCPoint4[27052] = {X 0.1632, Y 23.3903, Z -6.3333, A 0.000, B 0.000, C 0.000 }
gfCNCPoint4[27053] = {X -0.4341, Y 22.7068, Z -6.3333, A 0.000, B 0.000, C 0.000 }
gfCNCPoint4[27054] = {X -0.8722, Y 21.9118, Z -6.3333, A 0.000, B 0.000, C 0.000 }
gfCNCPoint4[27055] = {X -3.5467, Y 15.3561, Z -6.3333, A 0.000, B 0.000, C 0.000 }
gfCNCPoint4[27056] = {X -3.6292, Y 15.1115, Z -6.3333, A 0.000, B 0.000, C 0.000 }
gfCNCPoint4[27057] = {X -3.6966, Y 14.8624, Z -6.3333, A 0.000, B 0.000, C 0.000 }
gfCNCPoint4[27058] = {X -4.6242, Y 10.9714, Z -6.3333, A 0.000, B 0.000, C 0.000 }
gfCNCPoint4[27059] = {X -7.6966, Y 10.9714, Z -6.3333, A 0.000, B 0.000, C 0.000 }
gfCNCPoint4[27060] = {X -7.6966, Y 10.9714, Z -3.3333, A 0.000, B 0.000, C 0.000 }
gfCNCPoint4[27061] = {X -7.6966, Y 10.9714, Z 11.0000, A 0.000, B 0.000, C 0.000 }
gfCNCPoint4[27062] = {X -8.0051, Y 35.5750, Z 11.0000, A 0.000, B 0.000, C 0.000 }
gfCNCPoint4[27063] = {X -8.0051, Y 35.5750, Z -3.3333, A 0.000, B 0.000, C 0.000 }
gfCNCPoint4[27064] = {X -8.0051, Y 35.5750, Z -6.3333, A 0.000, B 0.000, C 0.000 }
gfCNCPoint4[27065] = {X -4.7015, Y 35.5337, Z -6.3333, A 0.000, B 0.000, C 0.000 }
gfCNCPoint4[27066] = {X -3.6966, Y 31.6619, Z -6.3333, A 0.000, B 0.000, C 0.000 }
gfCNCPoint4[27067] = {X -3.5879, Y 31.2658, Z -6.3333, A 0.000, B 0.000, C 0.000 }
gfCNCPoint4[27068] = {X -3.4681, Y 30.8729, Z -6.3333, A 0.000, B 0.000, C 0.000 }
gfCNCPoint4[27069] = {X -3.2953, Y 30.3656, Z -6.3333, A 0.000, B 0.000, C 0.000 }
gfCNCPoint4[27070] = {X -3.1041, Y 29.8650, Z -6.3333, A 0.000, B 0.000, C 0.000 }
gfCNCPoint4[27071] = {X -2.4949, Y 28.5733, Z -6.3333, A 0.000, B 0.000, C 0.000 }
gfCNCPoint4[27072] = {X -1.7185, Y 27.3747, Z -6.3333, A 0.000, B 0.000, C 0.000 }
gfCNCPoint4[27073] = {X -0.7889, Y 26.2905, Z -6.3333, A 0.000, B 0.000, C 0.000 }
gfCNCPoint4[27074] = {X 0.2773, Y 25.3402, Z -6.3333, A 0.000, B 0.000, C 0.000 }
gfCNCPoint4[27075] = {X 1.4609, Y 24.5410, Z -6.3333, A 0.000, B 0.000, C 0.000 }
gfCNCPoint4[27076] = {X 1.6935, Y 24.4095, Z -6.3333, A 0.000, B 0.000, C 0.000 }
gfCNCPoint4[27077] = {X 1.9293, Y 24.2840, Z -6.3333, A 0.000, B 0.000, C 0.000 }
gfCNCPoint4[27078] = {X 1.0588, Y 23.9332, Z -6.3333, A 0.000, B 0.000, C 0.000 }
gfCNCPoint4[27079] = {X 0.2891, Y 23.3962, Z -6.3333, A 0.000, B 0.000, C 0.000 }
gfCNCPoint4[27080] = {X -0.3407, Y 22.7003, Z -6.3333, A 0.000, B 0.000, C 0.000 }
gfCNCPoint4[27081] = {X -0.7984, Y 21.8809, Z -6.3333, A 0.000, B 0.000, C 0.000 }
gfCNCPoint4[27082] = {X -3.4717, Y 15.3282, Z -6.3333, A 0.000, B 0.000, C 0.000 }
gfCNCPoint4[27083] = {X -3.6097, Y 14.8815, Z -6.3333, A 0.000, B 0.000, C 0.000 }
gfCNCPoint4[27084] = {X -3.6966, Y 14.4221, Z -6.3333, A 0.000, B 0.000, C 0.000 }
gfCNCPoint4[27085] = {X -4.2187, Y 10.4563, Z -6.3333, A 0.000, B 0.000, C 0.000 }
gfCNCPoint4[27086] = {X -7.6966, Y 10.4563, Z -6.3333, A 0.000, B 0.000, C 0.000 }
gfCNCPoint4[27087] = {X -7.6966, Y 10.4563, Z -3.3333, A 0.000, B 0.000, C 0.000 }
gfCNCPoint4[27088] = {X -7.6966, Y 10.4563, Z 11.0000, A 0.000, B 0.000, C 0.000 }
gfCNCPoint4[27089] = {X -7.9946, Y 36.0092, Z 11.0000, A 0.000, B 0.000, C 0.000 }
gfCNCPoint4[27090] = {X -7.9946, Y 36.0092, Z -3.3333, A 0.000, B 0.000, C 0.000 }
gfCNCPoint4[27091] = {X -7.9946, Y 36.0092, Z -6.3333, A 0.000, B 0.000, C 0.000 }
gfCNCPoint4[27092] = {X -4.6157, Y 35.8875, Z -6.3333, A 0.000, B 0.000, C 0.000 }
gfCNCPoint4[27093] = {X -3.6966, Y 31.9945, Z -6.3333, A 0.000, B 0.000, C 0.000 }
gfCNCPoint4[27094] = {X -3.5550, Y 31.4429, Z -6.3333, A 0.000, B 0.000, C 0.000 }
gfCNCPoint4[27095] = {X -3.3919, Y 30.8973, Z -6.3333, A 0.000, B 0.000, C 0.000 }
gfCNCPoint4[27096] = {X -3.2200, Y 30.3926, Z -6.3333, A 0.000, B 0.000, C 0.000 }
gfCNCPoint4[27097] = {X -3.0298, Y 29.8946, Z -6.3333, A 0.000, B 0.000, C 0.000 }
gfCNCPoint4[27098] = {X -2.4251, Y 28.6125, Z -6.3333, A 0.000, B 0.000, C 0.000 }
gfCNCPoint4[27099] = {X -1.6545, Y 27.4227, Z -6.3333, A 0.000, B 0.000, C 0.000 }
gfCNCPoint4[27100] = {X -0.7318, Y 26.3466, Z -6.3333, A 0.000, B 0.000, C 0.000 }
gfCNCPoint4[27101] = {X 0.3264, Y 25.4034, Z -6.3333, A 0.000, B 0.000, C 0.000 }
gfCNCPoint4[27102] = {X 1.5011, Y 24.6101, Z -6.3333, A 0.000, B 0.000, C 0.000 }
gfCNCPoint4[27103] = {X 1.8264, Y 24.4285, Z -6.3333, A 0.000, B 0.000, C 0.000 }
gfCNCPoint4[27104] = {X 2.1578, Y 24.2584, Z -6.3333, A 0.000, B 0.000, C 0.000 }
gfCNCPoint4[27105] = {X 1.2392, Y 23.9363, Z -6.3333, A 0.000, B 0.000, C 0.000 }
gfCNCPoint4[27106] = {X 0.4230, Y 23.4056, Z -6.3333, A 0.000, B 0.000, C 0.000 }
gfCNCPoint4[27107] = {X -0.2443, Y 22.6968, Z -6.3333, A 0.000, B 0.000, C 0.000 }
gfCNCPoint4[27108] = {X -0.7246, Y 21.8500, Z -6.3333, A 0.000, B 0.000, C 0.000 }
gfCNCPoint4[27109] = {X -3.3967, Y 15.3004, Z -6.3333, A 0.000, B 0.000, C 0.000 }
gfCNCPoint4[27110] = {X -3.6236, Y 14.3619, Z -6.3333, A 0.000, B 0.000, C 0.000 }
gfCNCPoint4[27111] = {X -3.6236, Y 13.3964, Z -6.3333, A 0.000, B 0.000, C 0.000 }
gfCNCPoint4[27112] = {X -3.3967, Y 12.4579, Z -6.3333, A 0.000, B 0.000, C 0.000 }
gfCNCPoint4[27113] = {X -2.9670, Y 11.6160, Z -6.3333, A 0.000, B 0.000, C 0.000 }
gfCNCPoint4[27114] = {X -2.3552, Y 10.8956, Z -6.3333, A 0.000, B 0.000, C 0.000 }
gfCNCPoint4[27115] = {X -1.5940, Y 10.3353, Z -6.3333, A 0.000, B 0.000, C 0.000 }
gfCNCPoint4[27116] = {X -0.9967, Y 9.9945, Z -6.3333, A 0.000, B 0.000, C 0.000 }
gfCNCPoint4[27117] = {X -0.1385, Y 9.6278, Z -6.3333, A 0.000, B 0.000, C 0.000 }
gfCNCPoint4[27118] = {X 0.7806, Y 9.4658, Z -6.3333, A 0.000, B 0.000, C 0.000 }
gfCNCPoint4[27119] = {X 1.7125, Y 9.5168, Z -6.3333, A 0.000, B 0.000, C 0.000 }
gfCNCPoint4[27120] = {X 2.6085, Y 9.7783, Z -6.3333, A 0.000, B 0.000, C 0.000 }
gfCNCPoint4[27121] = {X 3.5852, Y 9.3395, Z -6.3333, A 0.000, B 0.000, C 0.000 }
gfCNCPoint4[27122] = {X 5.6410, Y 8.5650, Z -6.3333, A 0.000, B 0.000, C 0.000 }
gfCNCPoint4[27123] = {X 7.7600, Y 7.9854, Z -6.3333, A 0.000, B 0.000, C 0.000 }
gfCNCPoint4[27124] = {X 9.9238, Y 7.6056, Z -6.3333, A 0.000, B 0.000, C 0.000 }
gfCNCPoint4[27125] = {X 12.1135, Y 7.4290, Z -6.3333, A 0.000, B 0.000, C 0.000 }
gfCNCPoint4[27126] = {X 14.3102, Y 7.4570, Z -6.3333, A 0.000, B 0.000, C 0.000 }
gfCNCPoint4[27127] = {X 16.4947, Y 7.6895, Z -6.3333, A 0.000, B 0.000, C 0.000 }
gfCNCPoint4[27128] = {X 18.2062, Y 8.0401, Z -6.3333, A 0.000, B 0.000, C 0.000 }
gfCNCPoint4[27129] = {X 19.8735, Y 8.5624, Z -6.3333, A 0.000, B 0.000, C 0.000 }
gfCNCPoint4[27130] = {X 21.4791, Y 9.2510, Z -6.3333, A 0.000, B 0.000, C 0.000 }
gfCNCPoint4[27131] = {X 23.0067, Y 10.0990, Z -6.3333, A 0.000, B 0.000, C 0.000 }
gfCNCPoint4[27132] = {X 24.4404, Y 11.0974, Z -6.3333, A 0.000, B 0.000, C 0.000 }
gfCNCPoint4[27133] = {X 25.5054, Y 12.0287, Z -6.3333, A 0.000, B 0.000, C 0.000 }
gfCNCPoint4[27134] = {X 26.4609, Y 13.0723, Z -6.3333, A 0.000, B 0.000, C 0.000 }
gfCNCPoint4[27135] = {X 27.2949, Y 14.2151, Z -6.3333, A 0.000, B 0.000, C 0.000 }
gfCNCPoint4[27136] = {X 27.9973, Y 15.4433, Z -6.3333, A 0.000, B 0.000, C 0.000 }
gfCNCPoint4[27137] = {X 28.5594, Y 16.7417, Z -6.3333, A 0.000, B 0.000, C 0.000 }
gfCNCPoint4[27138] = {X 29.0262, Y 18.3710, Z -6.3333, A 0.000, B 0.000, C 0.000 }
gfCNCPoint4[27139] = {X 29.3032, Y 20.0430, Z -6.3333, A 0.000, B 0.000, C 0.000 }
gfCNCPoint4[27140] = {X 29.3866, Y 21.7358, Z -6.3333, A 0.000, B 0.000, C 0.000 }
gfCNCPoint4[27141] = {X 29.2755, Y 23.4270, Z -6.3333, A 0.000, B 0.000, C 0.000 }
gfCNCPoint4[27142] = {X 28.9711, Y 25.0943, Z -6.3333, A 0.000, B 0.000, C 0.000 }
gfCNCPoint4[27143] = {X 28.5034, Y 26.6013, Z -6.3333, A 0.000, B 0.000, C 0.000 }
gfCNCPoint4[27144] = {X 27.8329, Y 28.0298, Z -6.3333, A 0.000, B 0.000, C 0.000 }
gfCNCPoint4[27145] = {X 26.9725, Y 29.3525, Z -6.3333, A 0.000, B 0.000, C 0.000 }
gfCNCPoint4[27146] = {X 25.9384, Y 30.5445, Z -6.3333, A 0.000, B 0.000, C 0.000 }
gfCNCPoint4[27147] = {X 24.7503, Y 31.5829, Z -6.3333, A 0.000, B 0.000, C 0.000 }
gfCNCPoint4[27148] = {X 25.0472, Y 31.6500, Z -6.3333, A 0.000, B 0.000, C 0.000 }
gfCNCPoint4[27149] = {X 25.3383, Y 31.7390, Z -6.3333, A 0.000, B 0.000, C 0.000 }
gfCNCPoint4[27150] = {X 26.0575, Y 32.0700, Z -6.3333, A 0.000, B 0.000, C 0.000 }
gfCNCPoint4[27151] = {X 26.6992, Y 32.5336, Z -6.3333, A 0.000, B 0.000, C 0.000 }
gfCNCPoint4[27152] = {X 27.2393, Y 33.1123, Z -6.3333, A 0.000, B 0.000, C 0.000 }
gfCNCPoint4[27153] = {X 27.6575, Y 33.7845, Z -6.3333, A 0.000, B 0.000, C 0.000 }
gfCNCPoint4[27154] = {X 30.6940, Y 40.0576, Z -6.3333, A 0.000, B 0.000, C 0.000 }
gfCNCPoint4[27155] = {X 30.9967, Y 40.9162, Z -6.3333, A 0.000, B 0.000, C 0.000 }
gfCNCPoint4[27156] = {X 31.1015, Y 41.8206, Z -6.3333, A 0.000, B 0.000, C 0.000 }
gfCNCPoint4[27157] = {X 31.0032, Y 42.7257, Z -6.3333, A 0.000, B 0.000, C 0.000 }
gfCNCPoint4[27158] = {X 30.7066, Y 43.5864, Z -6.3333, A 0.000, B 0.000, C 0.000 }
gfCNCPoint4[27159] = {X 30.2265, Y 44.3600, Z -6.3333, A 0.000, B 0.000, C 0.000 }
gfCNCPoint4[27160] = {X 29.5868, Y 45.0078, Z -6.3333, A 0.000, B 0.000, C 0.000 }
gfCNCPoint4[27161] = {X 29.0508, Y 45.4413, Z -6.3333, A 0.000, B 0.000, C 0.000 }
gfCNCPoint4[27162] = {X 28.3677, Y 45.8888, Z -6.3333, A 0.000, B 0.000, C 0.000 }
gfCNCPoint4[27163] = {X 27.6093, Y 46.1917, Z -6.3333, A 0.000, B 0.000, C 0.000 }
gfCNCPoint4[27164] = {X 26.8058, Y 46.3380, Z -6.3333, A 0.000, B 0.000, C 0.000 }
gfCNCPoint4[27165] = {X 25.9893, Y 46.3218, Z -6.3333, A 0.000, B 0.000, C 0.000 }
gfCNCPoint4[27166] = {X 25.1923, Y 46.1438, Z -6.3333, A 0.000, B 0.000, C 0.000 }
gfCNCPoint4[27167] = {X 23.3785, Y 47.1073, Z -6.3333, A 0.000, B 0.000, C 0.000 }
gfCNCPoint4[27168] = {X 21.5013, Y 47.9406, Z -6.3333, A 0.000, B 0.000, C 0.000 }
gfCNCPoint4[27169] = {X 19.5700, Y 48.6395, Z -6.3333, A 0.000, B 0.000, C 0.000 }
gfCNCPoint4[27170] = {X 17.6503, Y 49.1816, Z -6.3333, A 0.000, B 0.000, C 0.000 }
gfCNCPoint4[27171] = {X 15.6901, Y 49.5516, Z -6.3333, A 0.000, B 0.000, C 0.000 }
gfCNCPoint4[27172] = {X 13.7049, Y 49.7466, Z -6.3333, A 0.000, B 0.000, C 0.000 }
gfCNCPoint4[27173] = {X 11.7103, Y 49.7652, Z -6.3333, A 0.000, B 0.000, C 0.000 }
gfCNCPoint4[27174] = {X 9.7218, Y 49.6071, Z -6.3333, A 0.000, B 0.000, C 0.000 }
gfCNCPoint4[27175] = {X 7.7551, Y 49.2736, Z -6.3333, A 0.000, B 0.000, C 0.000 }
gfCNCPoint4[27176] = {X 5.8808, Y 48.7600, Z -6.3333, A 0.000, B 0.000, C 0.000 }
gfCNCPoint4[27177] = {X 4.0800, Y 48.0293, Z -6.3333, A 0.000, B 0.000, C 0.000 }
gfCNCPoint4[27178] = {X 2.3777, Y 47.0917, Z -6.3333, A 0.000, B 0.000, C 0.000 }
gfCNCPoint4[27179] = {X 0.7976, Y 45.9602, Z -6.3333, A 0.000, B 0.000, C 0.000 }
gfCNCPoint4[27180] = {X -0.3140, Y 44.9610, Z -6.3333, A 0.000, B 0.000, C 0.000 }
gfCNCPoint4[27181] = {X -1.3014, Y 43.8388, Z -6.3333, A 0.000, B 0.000, C 0.000 }
gfCNCPoint4[27182] = {X -2.1510, Y 42.6089, Z -6.3333, A 0.000, B 0.000, C 0.000 }
gfCNCPoint4[27183] = {X -2.8510, Y 41.2883, Z -6.3333, A 0.000, B 0.000, C 0.000 }
gfCNCPoint4[27184] = {X -3.3921, Y 39.8949, Z -6.3333, A 0.000, B 0.000, C 0.000 }
gfCNCPoint4[27185] = {X -3.5570, Y 39.3407, Z -6.3333, A 0.000, B 0.000, C 0.000 }
gfCNCPoint4[27186] = {X -3.6966, Y 38.7795, Z -6.3333, A 0.000, B 0.000, C 0.000 }
gfCNCPoint4[27187] = {X -4.5747, Y 34.8771, Z -6.3333, A 0.000, B 0.000, C 0.000 }
gfCNCPoint4[27188] = {X -7.9977, Y 34.7711, Z -6.3333, A 0.000, B 0.000, C 0.000 }
gfCNCPoint4[27189] = {X -7.9977, Y 34.7711, Z -3.3333, A 0.000, B 0.000, C 0.000 }
gfCNCPoint4[27190] = {X -7.9977, Y 34.7711, Z 11.0000, A 0.000, B 0.000, C 0.000 }
gfCNCPoint4[27191] = {X -7.9710, Y 36.4909, Z 11.0000, A 0.000, B 0.000, C 0.000 }
gfCNCPoint4[27192] = {X -7.9710, Y 36.4909, Z -3.3333, A 0.000, B 0.000, C 0.000 }
gfCNCPoint4[27193] = {X -7.9710, Y 36.4909, Z -6.3333, A 0.000, B 0.000, C 0.000 }
gfCNCPoint4[27194] = {X -4.5194, Y 36.2764, Z -6.3333, A 0.000, B 0.000, C 0.000 }
gfCNCPoint4[27195] = {X -3.6966, Y 32.3619, Z -6.3333, A 0.000, B 0.000, C 0.000 }
gfCNCPoint4[27196] = {X -3.5247, Y 31.6369, Z -6.3333, A 0.000, B 0.000, C 0.000 }
gfCNCPoint4[27197] = {X -3.3157, Y 30.9217, Z -6.3333, A 0.000, B 0.000, C 0.000 }
gfCNCPoint4[27198] = {X -3.1444, Y 30.4189, Z -6.3333, A 0.000, B 0.000, C 0.000 }
gfCNCPoint4[27199] = {X -2.9549, Y 29.9228, Z -6.3333, A 0.000, B 0.000, C 0.000 }
gfCNCPoint4[27200] = {X -2.3548, Y 28.6506, Z -6.3333, A 0.000, B 0.000, C 0.000 }
gfCNCPoint4[27201] = {X -1.5900, Y 27.4701, Z -6.3333, A 0.000, B 0.000, C 0.000 }
gfCNCPoint4[27202] = {X -0.6744, Y 26.4023, Z -6.3333, A 0.000, B 0.000, C 0.000 }
gfCNCPoint4[27203] = {X 0.3757, Y 25.4664, Z -6.3333, A 0.000, B 0.000, C 0.000 }
gfCNCPoint4[27204] = {X 1.5414, Y 24.6793, Z -6.3333, A 0.000, B 0.000, C 0.000 }
gfCNCPoint4[27205] = {X 1.9718, Y 24.4422, Z -6.3333, A 0.000, B 0.000, C 0.000 }
gfCNCPoint4[27206] = {X 2.4129, Y 24.2254, Z -6.3333, A 0.000, B 0.000, C 0.000 }
gfCNCPoint4[27207] = {X 1.6210, Y 24.0149, Z -6.3333, A 0.000, B 0.000, C 0.000 }
gfCNCPoint4[27208] = {X 0.8887, Y 23.6475, Z -6.3333, A 0.000, B 0.000, C 0.000 }
gfCNCPoint4[27209] = {X 0.2465, Y 23.1386, Z -6.3333, A 0.000, B 0.000, C 0.000 }
gfCNCPoint4[27210] = {X -0.2784, Y 22.5095, Z -6.3333, A 0.000, B 0.000, C 0.000 }
gfCNCPoint4[27211] = {X -0.6642, Y 21.7867, Z -6.3333, A 0.000, B 0.000, C 0.000 }
gfCNCPoint4[27212] = {X -3.2754, Y 15.3911, Z -6.3333, A 0.000, B 0.000, C 0.000 }
gfCNCPoint4[27213] = {X -3.2990, Y 15.3320, Z -6.3333, A 0.000, B 0.000, C 0.000 }
gfCNCPoint4[27214] = {X -3.3217, Y 15.2725, Z -6.3333, A 0.000, B 0.000, C 0.000 }
gfCNCPoint4[27215] = {X -3.5441, Y 14.3524, Z -6.3333, A 0.000, B 0.000, C 0.000 }
gfCNCPoint4[27216] = {X -3.5441, Y 13.4058, Z -6.3333, A 0.000, B 0.000, C 0.000 }
gfCNCPoint4[27217] = {X -3.3217, Y 12.4858, Z -6.3333, A 0.000, B 0.000, C 0.000 }
gfCNCPoint4[27218] = {X -2.9005, Y 11.6604, Z -6.3333, A 0.000, B 0.000, C 0.000 }
gfCNCPoint4[27219] = {X -2.3006, Y 10.9541, Z -6.3333, A 0.000, B 0.000, C 0.000 }
gfCNCPoint4[27220] = {X -1.5544, Y 10.4048, Z -6.3333, A 0.000, B 0.000, C 0.000 }
gfCNCPoint4[27221] = {X -0.9063, Y 10.0355, Z -6.3333, A 0.000, B 0.000, C 0.000 }
gfCNCPoint4[27222] = {X -0.1050, Y 9.7014, Z -6.3333, A 0.000, B 0.000, C 0.000 }
gfCNCPoint4[27223] = {X 0.7494, Y 9.5480, Z -6.3333, A 0.000, B 0.000, C 0.000 }
gfCNCPoint4[27224] = {X 1.6168, Y 9.5825, Z -6.3333, A 0.000, B 0.000, C 0.000 }
gfCNCPoint4[27225] = {X 2.4564, Y 9.8034, Z -6.3333, A 0.000, B 0.000, C 0.000 }
gfCNCPoint4[27226] = {X 2.5434, Y 9.8379, Z -6.3333, A 0.000, B 0.000, C 0.000 }
gfCNCPoint4[27227] = {X 2.6297, Y 9.8745, Z -6.3333, A 0.000, B 0.000, C 0.000 }
gfCNCPoint4[27228] = {X 2.6555, Y 9.8430, Z -6.3333, A 0.000, B 0.000, C 0.000 }
gfCNCPoint4[27229] = {X 3.6169, Y 9.4130, Z -6.3333, A 0.000, B 0.000, C 0.000 }
gfCNCPoint4[27230] = {X 5.6657, Y 8.6411, Z -6.3333, A 0.000, B 0.000, C 0.000 }
gfCNCPoint4[27231] = {X 7.7776, Y 8.0634, Z -6.3333, A 0.000, B 0.000, C 0.000 }
gfCNCPoint4[27232] = {X 9.9341, Y 7.6849, Z -6.3333, A 0.000, B 0.000, C 0.000 }
gfCNCPoint4[27233] = {X 12.1164, Y 7.5089, Z -6.3333, A 0.000, B 0.000, C 0.000 }
gfCNCPoint4[27234] = {X 14.3057, Y 7.5369, Z -6.3333, A 0.000, B 0.000, C 0.000 }
gfCNCPoint4[27235] = {X 16.4829, Y 7.7687, Z -6.3333, A 0.000, B 0.000, C 0.000 }
gfCNCPoint4[27236] = {X 18.1864, Y 8.1176, Z -6.3333, A 0.000, B 0.000, C 0.000 }
gfCNCPoint4[27237] = {X 19.8458, Y 8.6375, Z -6.3333, A 0.000, B 0.000, C 0.000 }
gfCNCPoint4[27238] = {X 21.4440, Y 9.3229, Z -6.3333, A 0.000, B 0.000, C 0.000 }
gfCNCPoint4[27239] = {X 22.9644, Y 10.1669, Z -6.3333, A 0.000, B 0.000, C 0.000 }
gfCNCPoint4[27240] = {X 24.3914, Y 11.1606, Z -6.3333, A 0.000, B 0.000, C 0.000 }
gfCNCPoint4[27241] = {X 25.4496, Y 12.0860, Z -6.3333, A 0.000, B 0.000, C 0.000 }
gfCNCPoint4[27242] = {X 26.3989, Y 13.1229, Z -6.3333, A 0.000, B 0.000, C 0.000 }
gfCNCPoint4[27243] = {X 27.2276, Y 14.2584, Z -6.3333, A 0.000, B 0.000, C 0.000 }
gfCNCPoint4[27244] = {X 27.9256, Y 15.4787, Z -6.3333, A 0.000, B 0.000, C 0.000 }
gfCNCPoint4[27245] = {X 28.4841, Y 16.7687, Z -6.3333, A 0.000, B 0.000, C 0.000 }
gfCNCPoint4[27246] = {X 28.9484, Y 18.3893, Z -6.3333, A 0.000, B 0.000, C 0.000 }
gfCNCPoint4[27247] = {X 29.2237, Y 20.0524, Z -6.3333, A 0.000, B 0.000, C 0.000 }
gfCNCPoint4[27248] = {X 29.3066, Y 21.7361, Z -6.3333, A 0.000, B 0.000, C 0.000 }
gfCNCPoint4[27249] = {X 29.1959, Y 23.4182, Z -6.3333, A 0.000, B 0.000, C 0.000 }
gfCNCPoint4[27250] = {X 28.8931, Y 25.0766, Z -6.3333, A 0.000, B 0.000, C 0.000 }
gfCNCPoint4[27251] = {X 28.4150, Y 26.6079, Z -6.3333, A 0.000, B 0.000, C 0.000 }
gfCNCPoint4[27252] = {X 27.7261, Y 28.0568, Z -6.3333, A 0.000, B 0.000, C 0.000 }
gfCNCPoint4[27253] = {X 26.8402, Y 29.3943, Z -6.3333, A 0.000, B 0.000, C 0.000 }
gfCNCPoint4[27254] = {X 25.7749, Y 30.5938, Z -6.3333, A 0.000, B 0.000, C 0.000 }
gfCNCPoint4[27255] = {X 24.5514, Y 31.6315, Z -6.3333, A 0.000, B 0.000, C 0.000 }
gfCNCPoint4[27256] = {X 24.9362, Y 31.7044, Z -6.3333, A 0.000, B 0.000, C 0.000 }
gfCNCPoint4[27257] = {X 25.3121, Y 31.8146, Z -6.3333, A 0.000, B 0.000, C 0.000 }
gfCNCPoint4[27258] = {X 26.0245, Y 32.1434, Z -6.3333, A 0.000, B 0.000, C 0.000 }
gfCNCPoint4[27259] = {X 26.6591, Y 32.6049, Z -6.3333, A 0.000, B 0.000, C 0.000 }
gfCNCPoint4[27260] = {X 27.1913, Y 33.1814, Z -6.3333, A 0.000, B 0.000, C 0.000 }
gfCNCPoint4[27261] = {X 27.6008, Y 33.8508, Z -6.3333, A 0.000, B 0.000, C 0.000 }
gfCNCPoint4[27262] = {X 30.6220, Y 40.0925, Z -6.3333, A 0.000, B 0.000, C 0.000 }
gfCNCPoint4[27263] = {X 30.9188, Y 40.9342, Z -6.3333, A 0.000, B 0.000, C 0.000 }
gfCNCPoint4[27264] = {X 31.0215, Y 41.8209, Z -6.3333, A 0.000, B 0.000, C 0.000 }
gfCNCPoint4[27265] = {X 30.9251, Y 42.7082, Z -6.3333, A 0.000, B 0.000, C 0.000 }
gfCNCPoint4[27266] = {X 30.6343, Y 43.5521, Z -6.3333, A 0.000, B 0.000, C 0.000 }
gfCNCPoint4[27267] = {X 30.1637, Y 44.3105, Z -6.3333, A 0.000, B 0.000, C 0.000 }
gfCNCPoint4[27268] = {X 29.5365, Y 44.9456, Z -6.3333, A 0.000, B 0.000, C 0.000 }
gfCNCPoint4[27269] = {X 29.0005, Y 45.3790, Z -6.3333, A 0.000, B 0.000, C 0.000 }
gfCNCPoint4[27270] = {X 28.3244, Y 45.8211, Z -6.3333, A 0.000, B 0.000, C 0.000 }
gfCNCPoint4[27271] = {X 27.5734, Y 46.1187, Z -6.3333, A 0.000, B 0.000, C 0.000 }
gfCNCPoint4[27272] = {X 26.7780, Y 46.2599, Z -6.3333, A 0.000, B 0.000, C 0.000 }
gfCNCPoint4[27273] = {X 25.9705, Y 46.2388, Z -6.3333, A 0.000, B 0.000, C 0.000 }
gfCNCPoint4[27274] = {X 25.1836, Y 46.0564, Z -6.3333, A 0.000, B 0.000, C 0.000 }
gfCNCPoint4[27275] = {X 25.1079, Y 46.1001, Z -6.3333, A 0.000, B 0.000, C 0.000 }
gfCNCPoint4[27276] = {X 25.0320, Y 46.1435, Z -6.3333, A 0.000, B 0.000, C 0.000 }
gfCNCPoint4[27277] = {X 23.2598, Y 47.0759, Z -6.3333, A 0.000, B 0.000, C 0.000 }
gfCNCPoint4[27278] = {X 21.4276, Y 47.8839, Z -6.3333, A 0.000, B 0.000, C 0.000 }
gfCNCPoint4[27279] = {X 19.5440, Y 48.5638, Z -6.3333, A 0.000, B 0.000, C 0.000 }
gfCNCPoint4[27280] = {X 17.6311, Y 49.1039, Z -6.3333, A 0.000, B 0.000, C 0.000 }
gfCNCPoint4[27281] = {X 15.6779, Y 49.4725, Z -6.3333, A 0.000, B 0.000, C 0.000 }
gfCNCPoint4[27282] = {X 13.6997, Y 49.6668, Z -6.3333, A 0.000, B 0.000, C 0.000 }
gfCNCPoint4[27283] = {X 11.7121, Y 49.6852, Z -6.3333, A 0.000, B 0.000, C 0.000 }
gfCNCPoint4[27284] = {X 9.7307, Y 49.5276, Z -6.3333, A 0.000, B 0.000, C 0.000 }
gfCNCPoint4[27285] = {X 7.7710, Y 49.1952, Z -6.3333, A 0.000, B 0.000, C 0.000 }
gfCNCPoint4[27286] = {X 5.9056, Y 48.6839, Z -6.3333, A 0.000, B 0.000, C 0.000 }
gfCNCPoint4[27287] = {X 4.1135, Y 47.9566, Z -6.3333, A 0.000, B 0.000, C 0.000 }
gfCNCPoint4[27288] = {X 2.4194, Y 47.0234, Z -6.3333, A 0.000, B 0.000, C 0.000 }
gfCNCPoint4[27289] = {X 0.8469, Y 45.8972, Z -6.3333, A 0.000, B 0.000, C 0.000 }
gfCNCPoint4[27290] = {X -0.2576, Y 44.9043, Z -6.3333, A 0.000, B 0.000, C 0.000 }
gfCNCPoint4[27291] = {X -1.2387, Y 43.7892, Z -6.3333, A 0.000, B 0.000, C 0.000 }
gfCNCPoint4[27292] = {X -2.0827, Y 42.5671, Z -6.3333, A 0.000, B 0.000, C 0.000 }
gfCNCPoint4[27293] = {X -2.7783, Y 41.2549, Z -6.3333, A 0.000, B 0.000, C 0.000 }
gfCNCPoint4[27294] = {X -3.3159, Y 39.8703, Z -6.3333, A 0.000, B 0.000, C 0.000 }
gfCNCPoint4[27295] = {X -3.5286, Y 39.1354, Z -6.3333, A 0.000, B 0.000, C 0.000 }
gfCNCPoint4[27296] = {X -3.6966, Y 38.3890, Z -6.3333, A 0.000, B 0.000, C 0.000 }
gfCNCPoint4[27297] = {X -4.4571, Y 34.4620, Z -6.3333, A 0.000, B 0.000, C 0.000 }
gfCNCPoint4[27298] = {X -7.9745, Y 34.2545, Z -6.3333, A 0.000, B 0.000, C 0.000 }
gfCNCPoint4[27299] = {X -7.9745, Y 34.2545, Z -3.3333, A 0.000, B 0.000, C 0.000 }
gfCNCPoint4[27300] = {X -7.9745, Y 34.2545, Z 11.0000, A 0.000, B 0.000, C 0.000 }
gfCNCPoint4[27301] = {X 39.8245, Y 26.3831, Z 11.0000, A 0.000, B 0.000, C 0.000 }
gfCNCPoint4[27302] = {X 39.8245, Y 26.3831, Z -3.3333, A 0.000, B 0.000, C 0.000 }
gfCNCPoint4[27303] = {X 39.8245, Y 26.3831, Z -6.3333, A 0.000, B 0.000, C 0.000 }
gfCNCPoint4[27304] = {X 43.6479, Y 27.8073, Z -6.3333, A 0.000, B 0.000, C 0.000 }
gfCNCPoint4[27305] = {X 48.2901, Y 15.3446, Z -6.3333, A 0.000, B 0.000, C 0.000 }
gfCNCPoint4[27306] = {X 47.9079, Y 14.6186, Z -6.3333, A 0.000, B 0.000, C 0.000 }
gfCNCPoint4[27307] = {X 47.6697, Y 13.8334, Z -6.3333, A 0.000, B 0.000, C 0.000 }
gfCNCPoint4[27308] = {X 47.5844, Y 13.0173, Z -6.3333, A 0.000, B 0.000, C 0.000 }
gfCNCPoint4[27309] = {X 47.5842, Y 12.1868, Z -6.3333, A 0.000, B 0.000, C 0.000 }
gfCNCPoint4[27310] = {X 47.6925, Y 11.2255, Z -6.3333, A 0.000, B 0.000, C 0.000 }
gfCNCPoint4[27311] = {X 48.0120, Y 10.3125, Z -6.3333, A 0.000, B 0.000, C 0.000 }
gfCNCPoint4[27312] = {X 48.5267, Y 9.4933, Z -6.3333, A 0.000, B 0.000, C 0.000 }
gfCNCPoint4[27313] = {X 49.2107, Y 8.8093, Z -6.3333, A 0.000, B 0.000, C 0.000 }
gfCNCPoint4[27314] = {X 50.0298, Y 8.2946, Z -6.3333, A 0.000, B 0.000, C 0.000 }
gfCNCPoint4[27315] = {X 50.9429, Y 7.9751, Z -6.3333, A 0.000, B 0.000, C 0.000 }
gfCNCPoint4[27316] = {X 51.9042, Y 7.8668, Z -6.3333, A 0.000, B 0.000, C 0.000 }
gfCNCPoint4[27317] = {X 59.6221, Y 7.8668, Z -6.3333, A 0.000, B 0.000, C 0.000 }
gfCNCPoint4[27318] = {X 60.5834, Y 7.9751, Z -6.3333, A 0.000, B 0.000, C 0.000 }
gfCNCPoint4[27319] = {X 61.4965, Y 8.2946, Z -6.3333, A 0.000, B 0.000, C 0.000 }
gfCNCPoint4[27320] = {X 62.3156, Y 8.8093, Z -6.3333, A 0.000, B 0.000, C 0.000 }
gfCNCPoint4[27321] = {X 62.9996, Y 9.4933, Z -6.3333, A 0.000, B 0.000, C 0.000 }
gfCNCPoint4[27322] = {X 63.5143, Y 10.3124, Z -6.3333, A 0.000, B 0.000, C 0.000 }
gfCNCPoint4[27323] = {X 63.8338, Y 11.2255, Z -6.3333, A 0.000, B 0.000, C 0.000 }
gfCNCPoint4[27324] = {X 63.9421, Y 12.1868, Z -6.3333, A 0.000, B 0.000, C 0.000 }
gfCNCPoint4[27325] = {X 63.9421, Y 12.9782, Z -6.3333, A 0.000, B 0.000, C 0.000 }
gfCNCPoint4[27326] = {X 63.8584, Y 13.8244, Z -6.3333, A 0.000, B 0.000, C 0.000 }
gfCNCPoint4[27327] = {X 63.6105, Y 14.6379, Z -6.3333, A 0.000, B 0.000, C 0.000 }
gfCNCPoint4[27328] = {X 63.2081, Y 15.3871, Z -6.3333, A 0.000, B 0.000, C 0.000 }
gfCNCPoint4[27329] = {X 63.4265, Y 15.9633, Z -6.3333, A 0.000, B 0.000, C 0.000 }
gfCNCPoint4[27330] = {X 66.2401, Y 23.4305, Z -6.3333, A 0.000, B 0.000, C 0.000 }
gfCNCPoint4[27331] = {X 72.2104, Y 39.5004, Z -6.3333, A 0.000, B 0.000, C 0.000 }
gfCNCPoint4[27332] = {X 72.5158, Y 40.2686, Z -6.3333, A 0.000, B 0.000, C 0.000 }
gfCNCPoint4[27333] = {X 73.3599, Y 40.7705, Z -6.3333, A 0.000, B 0.000, C 0.000 }
gfCNCPoint4[27334] = {X 74.0689, Y 41.4501, Z -6.3333, A 0.000, B 0.000, C 0.000 }
gfCNCPoint4[27335] = {X 74.6061, Y 42.2723, Z -6.3333, A 0.000, B 0.000, C 0.000 }
gfCNCPoint4[27336] = {X 74.9437, Y 43.1945, Z -6.3333, A 0.000, B 0.000, C 0.000 }
gfCNCPoint4[27337] = {X 75.0643, Y 44.1692, Z -6.3333, A 0.000, B 0.000, C 0.000 }
gfCNCPoint4[27338] = {X 75.0645, Y 45.0000, Z -6.3333, A 0.000, B 0.000, C 0.000 }
gfCNCPoint4[27339] = {X 74.9561, Y 45.9613, Z -6.3333, A 0.000, B 0.000, C 0.000 }
gfCNCPoint4[27340] = {X 74.6366, Y 46.8744, Z -6.3333, A 0.000, B 0.000, C 0.000 }
gfCNCPoint4[27341] = {X 74.1220, Y 47.6935, Z -6.3333, A 0.000, B 0.000, C 0.000 }
gfCNCPoint4[27342] = {X 73.4379, Y 48.3775, Z -6.3333, A 0.000, B 0.000, C 0.000 }
gfCNCPoint4[27343] = {X 72.6188, Y 48.8922, Z -6.3333, A 0.000, B 0.000, C 0.000 }
gfCNCPoint4[27344] = {X 71.7057, Y 49.2117, Z -6.3333, A 0.000, B 0.000, C 0.000 }
gfCNCPoint4[27345] = {X 70.7445, Y 49.3200, Z -6.3333, A 0.000, B 0.000, C 0.000 }
gfCNCPoint4[27346] = {X 64.1851, Y 49.3200, Z -6.3333, A 0.000, B 0.000, C 0.000 }
gfCNCPoint4[27347] = {X 63.2238, Y 49.2117, Z -6.3333, A 0.000, B 0.000, C 0.000 }
gfCNCPoint4[27348] = {X 62.3108, Y 48.8922, Z -6.3333, A 0.000, B 0.000, C 0.000 }
gfCNCPoint4[27349] = {X 61.4917, Y 48.3775, Z -6.3333, A 0.000, B 0.000, C 0.000 }
gfCNCPoint4[27350] = {X 60.8076, Y 47.6935, Z -6.3333, A 0.000, B 0.000, C 0.000 }
gfCNCPoint4[27351] = {X 60.2929, Y 46.8744, Z -6.3333, A 0.000, B 0.000, C 0.000 }
gfCNCPoint4[27352] = {X 59.9734, Y 45.9613, Z -6.3333, A 0.000, B 0.000, C 0.000 }
gfCNCPoint4[27353] = {X 59.8651, Y 45.0000, Z -6.3333, A 0.000, B 0.000, C 0.000 }
gfCNCPoint4[27354] = {X 59.8651, Y 44.2085, Z -6.3333, A 0.000, B 0.000, C 0.000 }
gfCNCPoint4[27355] = {X 59.9517, Y 43.3502, Z -6.3333, A 0.000, B 0.000, C 0.000 }
gfCNCPoint4[27356] = {X 60.2071, Y 42.5262, Z -6.3333, A 0.000, B 0.000, C 0.000 }
gfCNCPoint4[27357] = {X 60.6210, Y 41.7694, Z -6.3333, A 0.000, B 0.000, C 0.000 }
gfCNCPoint4[27358] = {X 60.0066, Y 40.0892, Z -6.3333, A 0.000, B 0.000, C 0.000 }
gfCNCPoint4[27359] = {X 52.0779, Y 40.0892, Z -6.3333, A 0.000, B 0.000, C 0.000 }
gfCNCPoint4[27360] = {X 51.3349, Y 42.0855, Z -6.3333, A 0.000, B 0.000, C 0.000 }
gfCNCPoint4[27361] = {X 51.3379, Y 42.0905, Z -6.3333, A 0.000, B 0.000, C 0.000 }
gfCNCPoint4[27362] = {X 51.6391, Y 42.7498, Z -6.3333, A 0.000, B 0.000, C 0.000 }
gfCNCPoint4[27363] = {X 51.8258, Y 43.4502, Z -6.3333, A 0.000, B 0.000, C 0.000 }
gfCNCPoint4[27364] = {X 51.8928, Y 44.1720, Z -6.3333, A 0.000, B 0.000, C 0.000 }
gfCNCPoint4[27365] = {X 51.8929, Y 45.0000, Z -6.3333, A 0.000, B 0.000, C 0.000 }
gfCNCPoint4[27366] = {X 51.7846, Y 45.9613, Z -6.3333, A 0.000, B 0.000, C 0.000 }
gfCNCPoint4[27367] = {X 51.4651, Y 46.8744, Z -6.3333, A 0.000, B 0.000, C 0.000 }
gfCNCPoint4[27368] = {X 50.9504, Y 47.6935, Z -6.3333, A 0.000, B 0.000, C 0.000 }
gfCNCPoint4[27369] = {X 50.2664, Y 48.3775, Z -6.3333, A 0.000, B 0.000, C 0.000 }
gfCNCPoint4[27370] = {X 49.4473, Y 48.8922, Z -6.3333, A 0.000, B 0.000, C 0.000 }
gfCNCPoint4[27371] = {X 48.5342, Y 49.2117, Z -6.3333, A 0.000, B 0.000, C 0.000 }
gfCNCPoint4[27372] = {X 47.5729, Y 49.3200, Z -6.3333, A 0.000, B 0.000, C 0.000 }
gfCNCPoint4[27373] = {X 40.6393, Y 49.3200, Z -6.3333, A 0.000, B 0.000, C 0.000 }
gfCNCPoint4[27374] = {X 39.6780, Y 49.2117, Z -6.3333, A 0.000, B 0.000, C 0.000 }
gfCNCPoint4[27375] = {X 38.7649, Y 48.8922, Z -6.3333, A 0.000, B 0.000, C 0.000 }
gfCNCPoint4[27376] = {X 37.9458, Y 48.3775, Z -6.3333, A 0.000, B 0.000, C 0.000 }
gfCNCPoint4[27377] = {X 37.2618, Y 47.6935, Z -6.3333, A 0.000, B 0.000, C 0.000 }
gfCNCPoint4[27378] = {X 36.7471, Y 46.8744, Z -6.3333, A 0.000, B 0.000, C 0.000 }
gfCNCPoint4[27379] = {X 36.4276, Y 45.9613, Z -6.3333, A 0.000, B 0.000, C 0.000 }
gfCNCPoint4[27380] = {X 36.3193, Y 45.0000, Z -6.3333, A 0.000, B 0.000, C 0.000 }
gfCNCPoint4[27381] = {X 36.3193, Y 44.2086, Z -6.3333, A 0.000, B 0.000, C 0.000 }
gfCNCPoint4[27382] = {X 36.4360, Y 43.2116, Z -6.3333, A 0.000, B 0.000, C 0.000 }
gfCNCPoint4[27383] = {X 36.7795, Y 42.2685, Z -6.3333, A 0.000, B 0.000, C 0.000 }
gfCNCPoint4[27384] = {X 37.3315, Y 41.4301, Z -6.3333, A 0.000, B 0.000, C 0.000 }
gfCNCPoint4[27385] = {X 38.0621, Y 40.7418, Z -6.3333, A 0.000, B 0.000, C 0.000 }
gfCNCPoint4[27386] = {X 38.9318, Y 40.2406, Z -6.3333, A 0.000, B 0.000, C 0.000 }
gfCNCPoint4[27387] = {X 39.5230, Y 38.8450, Z -6.3333, A 0.000, B 0.000, C 0.000 }
gfCNCPoint4[27388] = {X 40.0638, Y 37.4291, Z -6.3333, A 0.000, B 0.000, C 0.000 }
gfCNCPoint4[27389] = {X 43.6479, Y 27.8073, Z -6.3333, A 0.000, B 0.000, C 0.000 }
gfCNCPoint4[27390] = {X 39.8995, Y 26.4110, Z -6.3333, A 0.000, B 0.000, C 0.000 }
gfCNCPoint4[27391] = {X 43.7228, Y 27.8352, Z -6.3333, A 0.000, B 0.000, C 0.000 }
gfCNCPoint4[27392] = {X 48.3793, Y 15.3344, Z -6.3333, A 0.000, B 0.000, C 0.000 }
gfCNCPoint4[27393] = {X 47.9922, Y 14.6130, Z -6.3333, A 0.000, B 0.000, C 0.000 }
gfCNCPoint4[27394] = {X 47.7508, Y 13.8307, Z -6.3333, A 0.000, B 0.000, C 0.000 }
gfCNCPoint4[27395] = {X 47.6644, Y 13.0166, Z -6.3333, A 0.000, B 0.000, C 0.000 }
gfCNCPoint4[27396] = {X 47.6642, Y 12.1868, Z -6.3333, A 0.000, B 0.000, C 0.000 }
gfCNCPoint4[27397] = {X 47.7705, Y 11.2433, Z -6.3333, A 0.000, B 0.000, C 0.000 }
gfCNCPoint4[27398] = {X 48.0841, Y 10.3472, Z -6.3333, A 0.000, B 0.000, C 0.000 }
gfCNCPoint4[27399] = {X 48.5893, Y 9.5432, Z -6.3333, A 0.000, B 0.000, C 0.000 }
gfCNCPoint4[27400] = {X 49.2606, Y 8.8719, Z -6.3333, A 0.000, B 0.000, C 0.000 }
gfCNCPoint4[27401] = {X 50.0646, Y 8.3667, Z -6.3333, A 0.000, B 0.000, C 0.000 }
gfCNCPoint4[27402] = {X 50.9607, Y 8.0531, Z -6.3333, A 0.000, B 0.000, C 0.000 }
gfCNCPoint4[27403] = {X 51.9042, Y 7.9468, Z -6.3333, A 0.000, B 0.000, C 0.000 }
gfCNCPoint4[27404] = {X 59.6221, Y 7.9468, Z -6.3333, A 0.000, B 0.000, C 0.000 }
gfCNCPoint4[27405] = {X 60.5656, Y 8.0531, Z -6.3333, A 0.000, B 0.000, C 0.000 }
gfCNCPoint4[27406] = {X 61.4618, Y 8.3667, Z -6.3333, A 0.000, B 0.000, C 0.000 }
gfCNCPoint4[27407] = {X 62.2657, Y 8.8718, Z -6.3333, A 0.000, B 0.000, C 0.000 }
gfCNCPoint4[27408] = {X 62.9371, Y 9.5432, Z -6.3333, A 0.000, B 0.000, C 0.000 }
gfCNCPoint4[27409] = {X 63.4422, Y 10.3471, Z -6.3333, A 0.000, B 0.000, C 0.000 }
gfCNCPoint4[27410] = {X 63.7558, Y 11.2433, Z -6.3333, A 0.000, B 0.000, C 0.000 }
gfCNCPoint4[27411] = {X 63.8621, Y 12.1868, Z -6.3333, A 0.000, B 0.000, C 0.000 }
gfCNCPoint4[27412] = {X 63.8621, Y 12.9782, Z -6.3333, A 0.000, B 0.000, C 0.000 }
gfCNCPoint4[27413] = {X 63.7772, Y 13.8222, Z -6.3333, A 0.000, B 0.000, C 0.000 }
gfCNCPoint4[27414] = {X 63.5260, Y 14.6325, Z -6.3333, A 0.000, B 0.000, C 0.000 }
gfCNCPoint4[27415] = {X 63.1185, Y 15.3765, Z -6.3333, A 0.000, B 0.000, C 0.000 }
gfCNCPoint4[27416] = {X 63.3516, Y 15.9916, Z -6.3333, A 0.000, B 0.000, C 0.000 }
gfCNCPoint4[27417] = {X 66.1652, Y 23.4585, Z -6.3333, A 0.000, B 0.000, C 0.000 }
gfCNCPoint4[27418] = {X 72.1357, Y 39.5291, Z -6.3333, A 0.000, B 0.000, C 0.000 }
gfCNCPoint4[27419] = {X 72.4535, Y 40.3285, Z -6.3333, A 0.000, B 0.000, C 0.000 }
gfCNCPoint4[27420] = {X 73.2909, Y 40.8186, Z -6.3333, A 0.000, B 0.000, C 0.000 }
gfCNCPoint4[27421] = {X 73.9950, Y 41.4863, Z -6.3333, A 0.000, B 0.000, C 0.000 }
gfCNCPoint4[27422] = {X 74.5288, Y 42.2966, Z -6.3333, A 0.000, B 0.000, C 0.000 }
gfCNCPoint4[27423] = {X 74.8644, Y 43.2070, Z -6.3333, A 0.000, B 0.000, C 0.000 }
gfCNCPoint4[27424] = {X 74.9843, Y 44.1699, Z -6.3333, A 0.000, B 0.000, C 0.000 }
gfCNCPoint4[27425] = {X 74.9845, Y 45.0000, Z -6.3333, A 0.000, B 0.000, C 0.000 }
gfCNCPoint4[27426] = {X 74.8782, Y 45.9435, Z -6.3333, A 0.000, B 0.000, C 0.000 }
gfCNCPoint4[27427] = {X 74.5646, Y 46.8397, Z -6.3333, A 0.000, B 0.000, C 0.000 }
gfCNCPoint4[27428] = {X 74.0594, Y 47.6436, Z -6.3333, A 0.000, B 0.000, C 0.000 }
gfCNCPoint4[27429] = {X 73.3881, Y 48.3150, Z -6.3333, A 0.000, B 0.000, C 0.000 }
gfCNCPoint4[27430] = {X 72.5841, Y 48.8201, Z -6.3333, A 0.000, B 0.000, C 0.000 }
gfCNCPoint4[27431] = {X 71.6879, Y 49.1337, Z -6.3333, A 0.000, B 0.000, C 0.000 }
gfCNCPoint4[27432] = {X 70.7445, Y 49.2400, Z -6.3333, A 0.000, B 0.000, C 0.000 }
gfCNCPoint4[27433] = {X 64.1851, Y 49.2400, Z -6.3333, A 0.000, B 0.000, C 0.000 }
gfCNCPoint4[27434] = {X 63.2416, Y 49.1337, Z -6.3333, A 0.000, B 0.000, C 0.000 }
gfCNCPoint4[27435] = {X 62.3455, Y 48.8201, Z -6.3333, A 0.000, B 0.000, C 0.000 }
gfCNCPoint4[27436] = {X 61.5415, Y 48.3150, Z -6.3333, A 0.000, B 0.000, C 0.000 }
gfCNCPoint4[27437] = {X 60.8702, Y 47.6436, Z -6.3333, A 0.000, B 0.000, C 0.000 }
gfCNCPoint4[27438] = {X 60.3650, Y 46.8397, Z -6.3333, A 0.000, B 0.000, C 0.000 }
gfCNCPoint4[27439] = {X 60.0514, Y 45.9435, Z -6.3333, A 0.000, B 0.000, C 0.000 }
gfCNCPoint4[27440] = {X 59.9451, Y 45.0000, Z -6.3333, A 0.000, B 0.000, C 0.000 }
gfCNCPoint4[27441] = {X 59.9451, Y 44.2085, Z -6.3333, A 0.000, B 0.000, C 0.000 }
gfCNCPoint4[27442] = {X 60.0328, Y 43.3527, Z -6.3333, A 0.000, B 0.000, C 0.000 }
gfCNCPoint4[27443] = {X 60.2915, Y 42.5323, Z -6.3333, A 0.000, B 0.000, C 0.000 }
gfCNCPoint4[27444] = {X 60.7104, Y 41.7809, Z -6.3333, A 0.000, B 0.000, C 0.000 }
gfCNCPoint4[27445] = {X 60.0626, Y 40.0092, Z -6.3333, A 0.000, B 0.000, C 0.000 }
gfCNCPoint4[27446] = {X 52.0223, Y 40.0092, Z -6.3333, A 0.000, B 0.000, C 0.000 }
gfCNCPoint4[27447] = {X 51.2466, Y 42.0934, Z -6.3333, A 0.000, B 0.000, C 0.000 }
gfCNCPoint4[27448] = {X 51.2687, Y 42.1305, Z -6.3333, A 0.000, B 0.000, C 0.000 }
gfCNCPoint4[27449] = {X 51.5640, Y 42.7774, Z -6.3333, A 0.000, B 0.000, C 0.000 }
gfCNCPoint4[27450] = {X 51.7471, Y 43.4646, Z -6.3333, A 0.000, B 0.000, C 0.000 }
gfCNCPoint4[27451] = {X 51.8128, Y 44.1726, Z -6.3333, A 0.000, B 0.000, C 0.000 }
gfCNCPoint4[27452] = {X 51.8129, Y 45.0000, Z -6.3333, A 0.000, B 0.000, C 0.000 }
gfCNCPoint4[27453] = {X 51.7066, Y 45.9435, Z -6.3333, A 0.000, B 0.000, C 0.000 }
gfCNCPoint4[27454] = {X 51.3930, Y 46.8397, Z -6.3333, A 0.000, B 0.000, C 0.000 }
gfCNCPoint4[27455] = {X 50.8879, Y 47.6436, Z -6.3333, A 0.000, B 0.000, C 0.000 }
gfCNCPoint4[27456] = {X 50.2165, Y 48.3150, Z -6.3333, A 0.000, B 0.000, C 0.000 }
gfCNCPoint4[27457] = {X 49.4126, Y 48.8201, Z -6.3333, A 0.000, B 0.000, C 0.000 }
gfCNCPoint4[27458] = {X 48.5164, Y 49.1337, Z -6.3333, A 0.000, B 0.000, C 0.000 }
gfCNCPoint4[27459] = {X 47.5729, Y 49.2400, Z -6.3333, A 0.000, B 0.000, C 0.000 }
gfCNCPoint4[27460] = {X 40.6393, Y 49.2400, Z -6.3333, A 0.000, B 0.000, C 0.000 }
gfCNCPoint4[27461] = {X 39.6958, Y 49.1337, Z -6.3333, A 0.000, B 0.000, C 0.000 }
gfCNCPoint4[27462] = {X 38.7996, Y 48.8201, Z -6.3333, A 0.000, B 0.000, C 0.000 }
gfCNCPoint4[27463] = {X 37.9957, Y 48.3150, Z -6.3333, A 0.000, B 0.000, C 0.000 }
gfCNCPoint4[27464] = {X 37.3243, Y 47.6436, Z -6.3333, A 0.000, B 0.000, C 0.000 }
gfCNCPoint4[27465] = {X 36.8192, Y 46.8397, Z -6.3333, A 0.000, B 0.000, C 0.000 }
gfCNCPoint4[27466] = {X 36.5056, Y 45.9435, Z -6.3333, A 0.000, B 0.000, C 0.000 }
gfCNCPoint4[27467] = {X 36.3993, Y 45.0000, Z -6.3333, A 0.000, B 0.000, C 0.000 }
gfCNCPoint4[27468] = {X 36.3993, Y 44.2086, Z -6.3333, A 0.000, B 0.000, C 0.000 }
gfCNCPoint4[27469] = {X 36.5152, Y 43.2240, Z -6.3333, A 0.000, B 0.000, C 0.000 }
gfCNCPoint4[27470] = {X 36.8566, Y 42.2933, Z -6.3333, A 0.000, B 0.000, C 0.000 }
gfCNCPoint4[27471] = {X 37.4048, Y 41.4673, Z -6.3333, A 0.000, B 0.000, C 0.000 }
gfCNCPoint4[27472] = {X 38.1298, Y 40.7912, Z -6.3333, A 0.000, B 0.000, C 0.000 }
gfCNCPoint4[27473] = {X 38.9920, Y 40.3019, Z -6.3333, A 0.000, B 0.000, C 0.000 }
gfCNCPoint4[27474] = {X 39.5913, Y 38.8895, Z -6.3333, A 0.000, B 0.000, C 0.000 }
gfCNCPoint4[27475] = {X 40.1390, Y 37.4563, Z -6.3333, A 0.000, B 0.000, C 0.000 }
gfCNCPoint4[27476] = {X 43.7228, Y 27.8352, Z -6.3333, A 0.000, B 0.000, C 0.000 }
gfCNCPoint4[27477] = {X 39.9744, Y 26.4389, Z -6.3333, A 0.000, B 0.000, C 0.000 }
gfCNCPoint4[27478] = {X 43.7978, Y 27.8631, Z -6.3333, A 0.000, B 0.000, C 0.000 }
gfCNCPoint4[27479] = {X 48.4687, Y 15.3238, Z -6.3333, A 0.000, B 0.000, C 0.000 }
gfCNCPoint4[27480] = {X 48.0765, Y 14.6072, Z -6.3333, A 0.000, B 0.000, C 0.000 }
gfCNCPoint4[27481] = {X 47.8320, Y 13.8279, Z -6.3333, A 0.000, B 0.000, C 0.000 }
gfCNCPoint4[27482] = {X 47.7444, Y 13.0158, Z -6.3333, A 0.000, B 0.000, C 0.000 }
gfCNCPoint4[27483] = {X 47.7442, Y 12.1868, Z -6.3333, A 0.000, B 0.000, C 0.000 }
gfCNCPoint4[27484] = {X 47.8485, Y 11.2611, Z -6.3333, A 0.000, B 0.000, C 0.000 }
gfCNCPoint4[27485] = {X 48.1562, Y 10.3819, Z -6.3333, A 0.000, B 0.000, C 0.000 }
gfCNCPoint4[27486] = {X 48.6518, Y 9.5931, Z -6.3333, A 0.000, B 0.000, C 0.000 }
gfCNCPoint4[27487] = {X 49.3105, Y 8.9344, Z -6.3333, A 0.000, B 0.000, C 0.000 }
gfCNCPoint4[27488] = {X 50.0993, Y 8.4388, Z -6.3333, A 0.000, B 0.000, C 0.000 }
gfCNCPoint4[27489] = {X 50.9785, Y 8.1311, Z -6.3333, A 0.000, B 0.000, C 0.000 }
gfCNCPoint4[27490] = {X 51.9042, Y 8.0268, Z -6.3333, A 0.000, B 0.000, C 0.000 }
gfCNCPoint4[27491] = {X 59.6221, Y 8.0268, Z -6.3333, A 0.000, B 0.000, C 0.000 }
gfCNCPoint4[27492] = {X 60.5478, Y 8.1311, Z -6.3333, A 0.000, B 0.000, C 0.000 }
gfCNCPoint4[27493] = {X 61.4271, Y 8.4388, Z -6.3333, A 0.000, B 0.000, C 0.000 }
gfCNCPoint4[27494] = {X 62.2158, Y 8.9344, Z -6.3333, A 0.000, B 0.000, C 0.000 }
gfCNCPoint4[27495] = {X 62.8745, Y 9.5931, Z -6.3333, A 0.000, B 0.000, C 0.000 }
gfCNCPoint4[27496] = {X 63.3702, Y 10.3819, Z -6.3333, A 0.000, B 0.000, C 0.000 }
gfCNCPoint4[27497] = {X 63.6778, Y 11.2611, Z -6.3333, A 0.000, B 0.000, C 0.000 }
gfCNCPoint4[27498] = {X 63.7821, Y 12.1868, Z -6.3333, A 0.000, B 0.000, C 0.000 }
gfCNCPoint4[27499] = {X 63.7821, Y 12.9782, Z -6.3333, A 0.000, B 0.000, C 0.000 }
gfCNCPoint4[27500] = {X 63.6960, Y 13.8199, Z -6.3333, A 0.000, B 0.000, C 0.000 }
gfCNCPoint4[27501] = {X 63.4414, Y 14.6268, Z -6.3333, A 0.000, B 0.000, C 0.000 }
gfCNCPoint4[27502] = {X 63.0288, Y 15.3655, Z -6.3333, A 0.000, B 0.000, C 0.000 }
gfCNCPoint4[27503] = {X 63.2768, Y 16.0199, Z -6.3333, A 0.000, B 0.000, C 0.000 }
gfCNCPoint4[27504] = {X 66.0903, Y 23.4865, Z -6.3333, A 0.000, B 0.000, C 0.000 }
gfCNCPoint4[27505] = {X 72.0610, Y 39.5578, Z -6.3333, A 0.000, B 0.000, C 0.000 }
gfCNCPoint4[27506] = {X 72.3913, Y 40.3886, Z -6.3333, A 0.000, B 0.000, C 0.000 }
gfCNCPoint4[27507] = {X 73.2219, Y 40.8670, Z -6.3333, A 0.000, B 0.000, C 0.000 }
gfCNCPoint4[27508] = {X 73.9210, Y 41.5227, Z -6.3333, A 0.000, B 0.000, C 0.000 }
gfCNCPoint4[27509] = {X 74.4515, Y 42.3210, Z -6.3333, A 0.000, B 0.000, C 0.000 }
gfCNCPoint4[27510] = {X 74.7851, Y 43.2196, Z -6.3333, A 0.000, B 0.000, C 0.000 }
gfCNCPoint4[27511] = {X 74.9043, Y 44.1706, Z -6.3333, A 0.000, B 0.000, C 0.000 }
gfCNCPoint4[27512] = {X 74.9045, Y 45.0000, Z -6.3333, A 0.000, B 0.000, C 0.000 }
gfCNCPoint4[27513] = {X 74.8002, Y 45.9257, Z -6.3333, A 0.000, B 0.000, C 0.000 }
gfCNCPoint4[27514] = {X 74.4925, Y 46.8050, Z -6.3333, A 0.000, B 0.000, C 0.000 }
gfCNCPoint4[27515] = {X 73.9969, Y 47.5937, Z -6.3333, A 0.000, B 0.000, C 0.000 }
gfCNCPoint4[27516] = {X 73.3382, Y 48.2524, Z -6.3333, A 0.000, B 0.000, C 0.000 }
gfCNCPoint4[27517] = {X 72.5494, Y 48.7480, Z -6.3333, A 0.000, B 0.000, C 0.000 }
gfCNCPoint4[27518] = {X 71.6701, Y 49.0557, Z -6.3333, A 0.000, B 0.000, C 0.000 }
gfCNCPoint4[27519] = {X 70.7445, Y 49.1600, Z -6.3333, A 0.000, B 0.000, C 0.000 }
gfCNCPoint4[27520] = {X 64.1851, Y 49.1600, Z -6.3333, A 0.000, B 0.000, C 0.000 }
gfCNCPoint4[27521] = {X 63.2594, Y 49.0557, Z -6.3333, A 0.000, B 0.000, C 0.000 }
gfCNCPoint4[27522] = {X 62.3802, Y 48.7480, Z -6.3333, A 0.000, B 0.000, C 0.000 }
gfCNCPoint4[27523] = {X 61.5914, Y 48.2524, Z -6.3333, A 0.000, B 0.000, C 0.000 }
gfCNCPoint4[27524] = {X 60.9327, Y 47.5937, Z -6.3333, A 0.000, B 0.000, C 0.000 }
gfCNCPoint4[27525] = {X 60.4371, Y 46.8050, Z -6.3333, A 0.000, B 0.000, C 0.000 }
gfCNCPoint4[27526] = {X 60.1294, Y 45.9257, Z -6.3333, A 0.000, B 0.000, C 0.000 }
gfCNCPoint4[27527] = {X 60.0251, Y 45.0000, Z -6.3333, A 0.000, B 0.000, C 0.000 }
gfCNCPoint4[27528] = {X 60.0251, Y 44.2086, Z -6.3333, A 0.000, B 0.000, C 0.000 }
gfCNCPoint4[27529] = {X 60.1140, Y 43.3554, Z -6.3333, A 0.000, B 0.000, C 0.000 }
gfCNCPoint4[27530] = {X 60.3760, Y 42.5385, Z -6.3333, A 0.000, B 0.000, C 0.000 }
gfCNCPoint4[27531] = {X 60.7999, Y 41.7928, Z -6.3333, A 0.000, B 0.000, C 0.000 }
gfCNCPoint4[27532] = {X 60.1185, Y 39.9292, Z -6.3333, A 0.000, B 0.000, C 0.000 }
gfCNCPoint4[27533] = {X 51.9667, Y 39.9292, Z -6.3333, A 0.000, B 0.000, C 0.000 }
gfCNCPoint4[27534] = {X 51.1583, Y 42.1014, Z -6.3333, A 0.000, B 0.000, C 0.000 }
gfCNCPoint4[27535] = {X 51.1994, Y 42.1706, Z -6.3333, A 0.000, B 0.000, C 0.000 }
gfCNCPoint4[27536] = {X 51.4889, Y 42.8050, Z -6.3333, A 0.000, B 0.000, C 0.000 }
gfCNCPoint4[27537] = {X 51.6684, Y 43.4789, Z -6.3333, A 0.000, B 0.000, C 0.000 }
gfCNCPoint4[27538] = {X 51.7328, Y 44.1733, Z -6.3333, A 0.000, B 0.000, C 0.000 }
gfCNCPoint4[27539] = {X 51.7329, Y 45.0000, Z -6.3333, A 0.000, B 0.000, C 0.000 }
gfCNCPoint4[27540] = {X 51.6286, Y 45.9257, Z -6.3333, A 0.000, B 0.000, C 0.000 }
gfCNCPoint4[27541] = {X 51.3210, Y 46.8050, Z -6.3333, A 0.000, B 0.000, C 0.000 }
gfCNCPoint4[27542] = {X 50.8253, Y 47.5937, Z -6.3333, A 0.000, B 0.000, C 0.000 }
gfCNCPoint4[27543] = {X 50.1666, Y 48.2524, Z -6.3333, A 0.000, B 0.000, C 0.000 }
gfCNCPoint4[27544] = {X 49.3779, Y 48.7480, Z -6.3333, A 0.000, B 0.000, C 0.000 }
gfCNCPoint4[27545] = {X 48.4986, Y 49.0557, Z -6.3333, A 0.000, B 0.000, C 0.000 }
gfCNCPoint4[27546] = {X 47.5729, Y 49.1600, Z -6.3333, A 0.000, B 0.000, C 0.000 }
gfCNCPoint4[27547] = {X 40.6393, Y 49.1600, Z -6.3333, A 0.000, B 0.000, C 0.000 }
gfCNCPoint4[27548] = {X 39.7136, Y 49.0557, Z -6.3333, A 0.000, B 0.000, C 0.000 }
gfCNCPoint4[27549] = {X 38.8343, Y 48.7480, Z -6.3333, A 0.000, B 0.000, C 0.000 }
gfCNCPoint4[27550] = {X 38.0456, Y 48.2524, Z -6.3333, A 0.000, B 0.000, C 0.000 }
gfCNCPoint4[27551] = {X 37.3869, Y 47.5937, Z -6.3333, A 0.000, B 0.000, C 0.000 }
gfCNCPoint4[27552] = {X 36.8913, Y 46.8050, Z -6.3333, A 0.000, B 0.000, C 0.000 }
gfCNCPoint4[27553] = {X 36.5836, Y 45.9257, Z -6.3333, A 0.000, B 0.000, C 0.000 }
gfCNCPoint4[27554] = {X 36.4793, Y 45.0000, Z -6.3333, A 0.000, B 0.000, C 0.000 }
gfCNCPoint4[27555] = {X 36.4793, Y 44.2086, Z -6.3333, A 0.000, B 0.000, C 0.000 }
gfCNCPoint4[27556] = {X 36.5945, Y 43.2365, Z -6.3333, A 0.000, B 0.000, C 0.000 }
gfCNCPoint4[27557] = {X 36.9337, Y 42.3182, Z -6.3333, A 0.000, B 0.000, C 0.000 }
gfCNCPoint4[27558] = {X 37.4781, Y 41.5047, Z -6.3333, A 0.000, B 0.000, C 0.000 }
gfCNCPoint4[27559] = {X 38.1975, Y 40.8408, Z -6.3333, A 0.000, B 0.000, C 0.000 }
gfCNCPoint4[27560] = {X 39.0522, Y 40.3635, Z -6.3333, A 0.000, B 0.000, C 0.000 }
gfCNCPoint4[27561] = {X 39.6596, Y 38.9341, Z -6.3333, A 0.000, B 0.000, C 0.000 }
gfCNCPoint4[27562] = {X 40.2142, Y 37.4835, Z -6.3333, A 0.000, B 0.000, C 0.000 }
gfCNCPoint4[27563] = {X 43.7978, Y 27.8631, Z -6.3333, A 0.000, B 0.000, C 0.000 }
gfCNCPoint4[27564] = {X 40.0494, Y 26.4668, Z -6.3333, A 0.000, B 0.000, C 0.000 }
gfCNCPoint4[27565] = {X 43.8728, Y 27.8910, Z -6.3333, A 0.000, B 0.000, C 0.000 }
gfCNCPoint4[27566] = {X 48.5582, Y 15.3126, Z -6.3333, A 0.000, B 0.000, C 0.000 }
gfCNCPoint4[27567] = {X 48.1610, Y 14.6012, Z -6.3333, A 0.000, B 0.000, C 0.000 }
gfCNCPoint4[27568] = {X 47.9131, Y 13.8250, Z -6.3333, A 0.000, B 0.000, C 0.000 }
gfCNCPoint4[27569] = {X 47.8244, Y 13.0151, Z -6.3333, A 0.000, B 0.000, C 0.000 }
gfCNCPoint4[27570] = {X 47.8242, Y 12.1868, Z -6.3333, A 0.000, B 0.000, C 0.000 }
gfCNCPoint4[27571] = {X 47.9265, Y 11.2789, Z -6.3333, A 0.000, B 0.000, C 0.000 }
gfCNCPoint4[27572] = {X 48.2283, Y 10.4166, Z -6.3333, A 0.000, B 0.000, C 0.000 }
gfCNCPoint4[27573] = {X 48.7144, Y 9.6430, Z -6.3333, A 0.000, B 0.000, C 0.000 }
gfCNCPoint4[27574] = {X 49.3604, Y 8.9969, Z -6.3333, A 0.000, B 0.000, C 0.000 }
gfCNCPoint4[27575] = {X 50.1340, Y 8.5109, Z -6.3333, A 0.000, B 0.000, C 0.000 }
gfCNCPoint4[27576] = {X 50.9963, Y 8.2091, Z -6.3333, A 0.000, B 0.000, C 0.000 }
gfCNCPoint4[27577] = {X 51.9042, Y 8.1068, Z -6.3333, A 0.000, B 0.000, C 0.000 }
gfCNCPoint4[27578] = {X 59.6221, Y 8.1068, Z -6.3333, A 0.000, B 0.000, C 0.000 }
gfCNCPoint4[27579] = {X 60.5300, Y 8.2091, Z -6.3333, A 0.000, B 0.000, C 0.000 }
gfCNCPoint4[27580] = {X 61.3924, Y 8.5109, Z -6.3333, A 0.000, B 0.000, C 0.000 }
gfCNCPoint4[27581] = {X 62.1660, Y 8.9969, Z -6.3333, A 0.000, B 0.000, C 0.000 }
gfCNCPoint4[27582] = {X 62.8120, Y 9.6430, Z -6.3333, A 0.000, B 0.000, C 0.000 }
gfCNCPoint4[27583] = {X 63.2981, Y 10.4166, Z -6.3333, A 0.000, B 0.000, C 0.000 }
gfCNCPoint4[27584] = {X 63.5998, Y 11.2789, Z -6.3333, A 0.000, B 0.000, C 0.000 }
gfCNCPoint4[27585] = {X 63.7021, Y 12.1868, Z -6.3333, A 0.000, B 0.000, C 0.000 }
gfCNCPoint4[27586] = {X 63.7021, Y 12.9782, Z -6.3333, A 0.000, B 0.000, C 0.000 }
gfCNCPoint4[27587] = {X 63.6148, Y 13.8175, Z -6.3333, A 0.000, B 0.000, C 0.000 }
gfCNCPoint4[27588] = {X 63.3567, Y 14.6209, Z -6.3333, A 0.000, B 0.000, C 0.000 }
gfCNCPoint4[27589] = {X 62.9389, Y 15.3540, Z -6.3333, A 0.000, B 0.000, C 0.000 }
gfCNCPoint4[27590] = {X 63.2020, Y 16.0481, Z -6.3333, A 0.000, B 0.000, C 0.000 }
